Yaskawa INFORM job: DEMO_ROOF_SIDE_0625_3PAINT_45.JBI

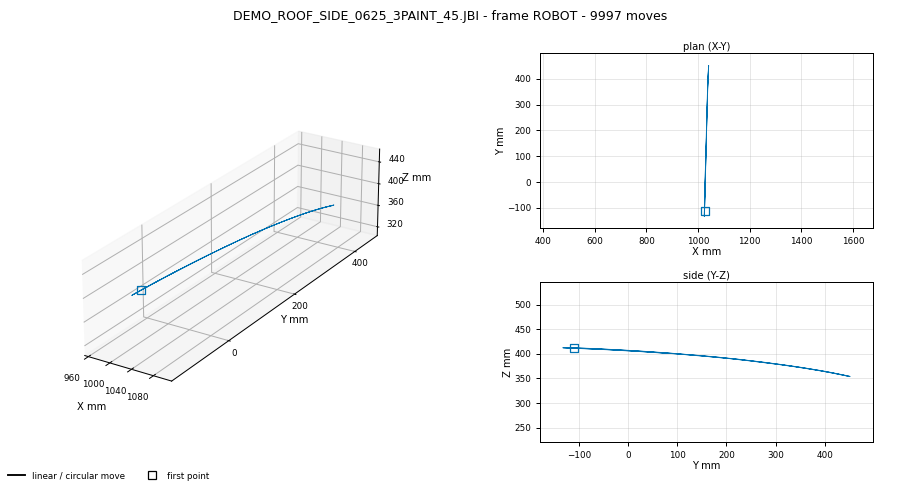
[picture p0: tool path of DEMO_ROOF_SIDE_0625_3PAINT_45.JBI in frame ROBOT, 9997 of 9997 moves have a stored position in this frame; points joined in program order, loops and branches not executed]
/JOB
//NAME DEMO_ROOF_SIDE_0625_3PAINT45
//POS
///NPOS 9997,0,0,0,0,0
///TOOL 0
///USER 0
///POSTYPE ROBOT
///RECTAN
///RCONF 1,0,0,0,0,0,0,0,0,0,0,0,0,0,0,0,0,0,0,0,0,0,0,0
C00000=1025.826,-110.558,412.586,166.562,45.746,158.343
C00001=1025.832,-110.309,412.577,166.564,45.743,158.343
C00002=1025.837,-110.058,412.568,166.568,45.740,158.343
C00003=1025.843,-109.809,412.559,166.570,45.738,158.343
C00004=1025.849,-109.559,412.550,166.574,45.735,158.343
C00005=1025.854,-109.310,412.541,166.577,45.732,158.343
C00006=1025.860,-109.059,412.532,166.579,45.729,158.343
C00007=1025.866,-108.810,412.523,166.583,45.726,158.342
C00008=1025.872,-108.560,412.514,166.586,45.724,158.342
C00009=1025.877,-108.311,412.505,166.589,45.721,158.342
C00010=1025.883,-108.060,412.496,166.592,45.718,158.342
C00011=1025.889,-107.811,412.487,166.594,45.716,158.342
C00012=1025.895,-107.561,412.478,166.598,45.713,158.342
C00013=1025.900,-107.312,412.469,166.601,45.710,158.342
C00014=1025.906,-107.061,412.460,166.604,45.708,158.341
C00015=1025.912,-106.812,412.450,166.607,45.705,158.341
C00016=1025.918,-106.562,412.442,166.609,45.703,158.341
C00017=1025.924,-106.312,412.432,166.613,45.700,158.341
C00018=1025.929,-106.063,412.423,166.616,45.697,158.341
C00019=1025.935,-105.812,412.414,166.618,45.694,158.341
C00020=1025.941,-105.563,412.405,166.622,45.692,158.341
C00021=1025.946,-105.313,412.395,166.624,45.689,158.340
C00022=1025.952,-105.063,412.386,166.628,45.686,158.340
C00023=1025.958,-104.814,412.377,166.630,45.684,158.340
C00024=1025.964,-104.564,412.367,166.634,45.681,158.340
C00025=1025.969,-104.314,412.359,166.637,45.678,158.340
C00026=1025.975,-104.064,412.349,166.640,45.676,158.340
C00027=1025.981,-103.814,412.339,166.643,45.673,158.340
C00028=1025.986,-103.565,412.330,166.645,45.670,158.340
C00029=1025.992,-103.315,412.321,166.649,45.668,158.340
C00030=1025.998,-103.066,412.312,166.651,45.665,158.339
C00031=1026.004,-102.816,412.302,166.654,45.662,158.339
C00032=1026.010,-102.566,412.293,166.658,45.659,158.339
C00033=1026.014,-102.316,412.283,166.660,45.657,158.339
C00034=1026.021,-102.066,412.274,166.664,45.654,158.339
C00035=1026.027,-101.817,412.264,166.666,45.652,158.339
C00036=1026.032,-101.567,412.255,166.670,45.649,158.339
C00037=1026.039,-101.281,412.244,166.673,45.646,158.338
C00038=1026.046,-100.994,412.233,166.676,45.643,158.338
C00039=1026.052,-100.708,412.223,166.679,45.640,158.338
C00040=1026.059,-100.422,412.211,166.683,45.637,158.338
C00041=1026.064,-100.173,412.203,166.686,45.634,158.338
C00042=1026.070,-99.923,412.193,166.690,45.631,158.338
C00043=1026.077,-99.673,412.184,166.692,45.629,158.337
C00044=1026.083,-99.423,412.174,166.696,45.626,158.337
C00045=1026.088,-99.174,412.164,166.698,45.624,158.337
C00046=1026.094,-98.924,412.155,166.701,45.621,158.337
C00047=1026.100,-98.674,412.145,166.704,45.619,158.337
C00048=1026.106,-98.424,412.136,166.707,45.616,158.337
C00049=1026.111,-98.175,412.127,166.711,45.613,158.337
C00050=1026.117,-97.925,412.117,166.713,45.610,158.336
C00051=1026.123,-97.675,412.107,166.716,45.608,158.336
C00052=1026.129,-97.425,412.098,166.719,45.605,158.336
C00053=1026.134,-97.176,412.088,166.722,45.603,158.336
C00054=1026.140,-96.926,412.078,166.725,45.600,158.336
C00055=1026.146,-96.676,412.068,166.728,45.598,158.336
C00056=1026.152,-96.426,412.059,166.731,45.595,158.336
C00057=1026.157,-96.176,412.049,166.734,45.593,158.336
C00058=1026.163,-95.927,412.039,166.737,45.590,158.336
C00059=1026.168,-95.677,412.028,166.740,45.588,158.336
C00060=1026.175,-95.427,412.019,166.742,45.585,158.335
C00061=1026.179,-95.178,412.009,166.746,45.583,158.335
C00062=1026.186,-94.928,411.999,166.748,45.580,158.335
C00063=1026.192,-94.678,411.990,166.752,45.577,158.335
C00064=1026.197,-94.428,411.980,166.754,45.575,158.335
C00065=1026.203,-94.178,411.970,166.758,45.572,158.335
C00066=1026.208,-93.929,411.960,166.760,45.570,158.335
C00067=1026.214,-93.679,411.951,166.764,45.567,158.334
C00068=1026.220,-93.430,411.940,166.766,45.565,158.334
C00069=1026.226,-93.180,411.930,166.770,45.562,158.334
C00070=1026.232,-92.930,411.920,166.772,45.560,158.334
C00071=1026.238,-92.680,411.911,166.775,45.557,158.334
C00072=1026.243,-92.431,411.901,166.778,45.555,158.334
C00073=1026.249,-92.182,411.891,166.781,45.552,158.334
C00074=1026.255,-91.931,411.880,166.785,45.550,158.334
C00075=1026.261,-91.682,411.871,166.787,45.547,158.334
C00076=1026.266,-91.431,411.861,166.791,45.545,158.334
C00077=1026.272,-91.182,411.851,166.793,45.542,158.333
C00078=1026.278,-90.932,411.840,166.797,45.539,158.333
C00079=1026.284,-90.682,411.831,166.799,45.537,158.333
C00080=1026.289,-90.433,411.821,166.802,45.534,158.333
C00081=1026.295,-90.183,411.811,166.805,45.532,158.333
C00082=1026.301,-89.934,411.800,166.808,45.529,158.333
C00083=1026.307,-89.684,411.791,166.811,45.527,158.333
C00084=1026.313,-89.434,411.781,166.814,45.524,158.332
C00085=1026.319,-89.185,411.770,166.817,45.522,158.332
C00086=1026.325,-88.935,411.760,166.820,45.519,158.332
C00087=1026.331,-88.685,411.751,166.823,45.516,158.332
C00088=1026.336,-88.435,411.740,166.826,45.514,158.332
C00089=1026.343,-88.185,411.730,166.828,45.512,158.332
C00090=1026.348,-87.935,411.720,166.832,45.509,158.332
C00091=1026.354,-87.686,411.710,166.834,45.507,158.332
C00092=1026.360,-87.436,411.700,166.838,45.504,158.332
C00093=1026.366,-87.186,411.690,166.840,45.502,158.331
C00094=1026.372,-86.937,411.679,166.844,45.499,158.331
C00095=1026.377,-86.687,411.669,166.846,45.497,158.331
C00096=1026.384,-86.437,411.659,166.850,45.494,158.331
C00097=1026.389,-86.187,411.649,166.852,45.492,158.331
C00098=1026.395,-85.938,411.639,166.856,45.489,158.331
C00099=1026.401,-85.688,411.628,166.858,45.487,158.331
C00100=1026.407,-85.438,411.619,166.861,45.484,158.330
C00101=1026.414,-85.154,411.607,166.865,45.481,158.330
C00102=1026.420,-84.871,411.596,166.868,45.478,158.330
C00103=1026.427,-84.586,411.584,166.871,45.475,158.330
C00104=1026.434,-84.303,411.572,166.875,45.472,158.330
C00105=1026.440,-84.053,411.562,166.877,45.470,158.330
C00106=1026.445,-83.803,411.551,166.881,45.467,158.330
C00107=1026.452,-83.554,411.542,166.884,45.465,158.330
C00108=1026.458,-83.303,411.531,166.887,45.462,158.329
C00109=1026.464,-83.054,411.521,166.890,45.459,158.329
C00110=1026.470,-82.804,411.510,166.893,45.457,158.329
C00111=1026.476,-82.554,411.501,166.896,45.454,158.329
C00112=1026.482,-82.305,411.490,166.899,45.452,158.329
C00113=1026.488,-82.055,411.480,166.902,45.449,158.329
C00114=1026.494,-81.806,411.469,166.904,45.446,158.328
C00115=1026.499,-81.556,411.459,166.908,45.444,158.328
C00116=1026.506,-81.306,411.449,166.910,45.441,158.328
C00117=1026.511,-81.056,411.439,166.914,45.439,158.328
C00118=1026.518,-80.806,411.428,166.916,45.436,158.328
C00119=1026.524,-80.557,411.417,166.919,45.433,158.328
C00120=1026.530,-80.307,411.408,166.922,45.431,158.328
C00121=1026.536,-80.058,411.397,166.925,45.428,158.328
C00122=1026.541,-79.807,411.386,166.928,45.426,158.327
C00123=1026.547,-79.558,411.376,166.931,45.424,158.327
C00124=1026.553,-79.309,411.365,166.934,45.421,158.327
C00125=1026.559,-79.058,411.355,166.937,45.419,158.327
C00126=1026.565,-78.808,411.344,166.940,45.417,158.327
C00127=1026.571,-78.559,411.333,166.943,45.414,158.327
C00128=1026.577,-78.310,411.322,166.946,45.412,158.327
C00129=1026.582,-78.059,411.312,166.948,45.410,158.327
C00130=1026.589,-77.810,411.302,166.952,45.407,158.326
C00131=1026.595,-77.560,411.290,166.954,45.405,158.326
C00132=1026.601,-77.311,411.280,166.958,45.402,158.326
C00133=1026.606,-77.061,411.269,166.960,45.400,158.326
C00134=1026.612,-76.811,411.259,166.963,45.397,158.326
C00135=1026.618,-76.561,411.248,166.966,45.395,158.326
C00136=1026.624,-76.312,411.237,166.970,45.392,158.326
C00137=1026.630,-76.062,411.226,166.972,45.390,158.326
C00138=1026.636,-75.813,411.215,166.976,45.387,158.326
C00139=1026.642,-75.562,411.205,166.978,45.385,158.325
C00140=1026.647,-75.313,411.194,166.980,45.383,158.325
C00141=1026.653,-75.064,411.183,166.984,45.380,158.325
C00142=1026.660,-74.814,411.173,166.986,45.378,158.325
C00143=1026.666,-74.564,411.162,166.990,45.375,158.325
C00144=1026.672,-74.315,411.151,166.992,45.373,158.325
C00145=1026.677,-74.065,411.140,166.996,45.371,158.325
C00146=1026.684,-73.815,411.129,166.998,45.368,158.325
C00147=1026.689,-73.565,411.119,167.001,45.366,158.324
C00148=1026.694,-73.315,411.107,167.004,45.364,158.324
C00149=1026.700,-73.066,411.096,167.007,45.362,158.324
C00150=1026.706,-72.815,411.085,167.009,45.359,158.324
C00151=1026.712,-72.566,411.074,167.013,45.357,158.324
C00152=1026.718,-72.316,411.063,167.016,45.355,158.324
C00153=1026.724,-72.068,411.052,167.019,45.352,158.324
C00154=1026.730,-71.817,411.040,167.021,45.350,158.324
C00155=1026.736,-71.568,411.030,167.024,45.348,158.324
C00156=1026.741,-71.318,411.018,167.028,45.345,158.324
C00157=1026.747,-71.068,411.007,167.030,45.343,158.323
C00158=1026.753,-70.818,410.996,167.033,45.341,158.323
C00159=1026.759,-70.569,410.985,167.036,45.338,158.323
C00160=1026.764,-70.319,410.974,167.039,45.336,158.323
C00161=1026.771,-70.069,410.963,167.042,45.333,158.323
C00162=1026.776,-69.820,410.952,167.045,45.331,158.323
C00163=1026.782,-69.570,410.941,167.047,45.329,158.323
C00164=1026.788,-69.320,410.929,167.051,45.326,158.323
C00165=1026.795,-69.039,410.917,167.054,45.324,158.323
C00166=1026.801,-68.757,410.904,167.056,45.322,158.323
C00167=1026.808,-68.475,410.892,167.060,45.319,158.322
C00168=1026.814,-68.193,410.879,167.063,45.316,158.322
C00169=1026.821,-67.944,410.867,167.066,45.314,158.322
C00170=1026.827,-67.694,410.857,167.069,45.311,158.322
C00171=1026.832,-67.445,410.846,167.072,45.309,158.322
C00172=1026.838,-67.194,410.834,167.075,45.307,158.322
C00173=1026.844,-66.945,410.823,167.078,45.305,158.322
C00174=1026.850,-66.695,410.811,167.080,45.302,158.322
C00175=1026.856,-66.445,410.800,167.084,45.300,158.322
C00176=1026.862,-66.196,410.789,167.087,45.298,158.322
C00177=1026.868,-65.946,410.778,167.089,45.296,158.321
C00178=1026.874,-65.697,410.766,167.093,45.293,158.321
C00179=1026.880,-65.446,410.755,167.095,45.291,158.321
C00180=1026.885,-65.197,410.744,167.097,45.289,158.321
C00181=1026.891,-64.947,410.733,167.101,45.286,158.321
C00182=1026.898,-64.698,410.721,167.104,45.284,158.321
C00183=1026.904,-64.448,410.710,167.107,45.281,158.321
C00184=1026.910,-64.198,410.699,167.110,45.279,158.321
C00185=1026.915,-63.949,410.687,167.112,45.277,158.320
C00186=1026.922,-63.699,410.675,167.116,45.274,158.320
C00187=1026.927,-63.449,410.664,167.118,45.272,158.320
C00188=1026.933,-63.200,410.653,167.121,45.270,158.320
C00189=1026.940,-62.950,410.642,167.124,45.268,158.320
C00190=1026.945,-62.700,410.630,167.127,45.266,158.320
C00191=1026.951,-62.451,410.618,167.130,45.263,158.320
C00192=1026.957,-62.201,410.607,167.133,45.261,158.320
C00193=1026.963,-61.951,410.596,167.135,45.259,158.320
C00194=1026.969,-61.702,410.584,167.138,45.256,158.319
C00195=1026.976,-61.452,410.573,167.141,45.254,158.319
C00196=1026.981,-61.202,410.562,167.144,45.252,158.319
C00197=1026.987,-60.953,410.550,167.147,45.249,158.319
C00198=1026.993,-60.703,410.539,167.150,45.247,158.319
C00199=1027.000,-60.454,410.527,167.152,45.245,158.319
C00200=1027.006,-60.204,410.516,167.156,45.242,158.319
C00201=1027.011,-59.954,410.503,167.158,45.240,158.319
C00202=1027.018,-59.704,410.492,167.162,45.238,158.319
C00203=1027.024,-59.455,410.481,167.164,45.235,158.318
C00204=1027.030,-59.205,410.469,167.167,45.233,158.318
C00205=1027.036,-58.956,410.459,167.170,45.230,158.318
C00206=1027.042,-58.706,410.446,167.173,45.228,158.318
C00207=1027.048,-58.456,410.435,167.175,45.226,158.318
C00208=1027.054,-58.207,410.423,167.178,45.223,158.318
C00209=1027.061,-57.956,410.412,167.181,45.221,158.318
C00210=1027.066,-57.707,410.400,167.185,45.219,158.318
C00211=1027.072,-57.457,410.388,167.187,45.216,158.317
C00212=1027.078,-57.208,410.377,167.190,45.214,158.317
C00213=1027.085,-56.958,410.366,167.193,45.211,158.317
C00214=1027.091,-56.708,410.354,167.195,45.209,158.317
C00215=1027.097,-56.459,410.341,167.198,45.207,158.317
C00216=1027.103,-56.209,410.330,167.201,45.204,158.317
C00217=1027.109,-55.960,410.319,167.204,45.202,158.317
C00218=1027.115,-55.710,410.307,167.207,45.199,158.316
C00219=1027.122,-55.460,410.295,167.210,45.197,158.316
C00220=1027.127,-55.211,410.284,167.213,45.195,158.316
C00221=1027.134,-54.961,410.272,167.216,45.192,158.316
C00222=1027.140,-54.712,410.260,167.218,45.190,158.316
C00223=1027.146,-54.462,410.249,167.221,45.188,158.316
C00224=1027.152,-54.212,410.237,167.224,45.185,158.316
C00225=1027.158,-53.962,410.225,167.227,45.183,158.316
C00226=1027.164,-53.713,410.214,167.229,45.181,158.315
C00227=1027.171,-53.464,410.202,167.233,45.179,158.315
C00228=1027.177,-53.213,410.190,167.235,45.176,158.315
C00229=1027.183,-52.933,410.177,167.239,45.174,158.315
C00230=1027.191,-52.652,410.164,167.242,45.171,158.315
C00231=1027.197,-52.372,410.150,167.246,45.168,158.315
C00232=1027.205,-52.091,410.137,167.248,45.165,158.315
C00233=1027.211,-51.842,410.126,167.252,45.163,158.314
C00234=1027.217,-51.592,410.114,167.254,45.160,158.314
C00235=1027.223,-51.342,410.101,167.256,45.158,158.314
C00236=1027.230,-51.092,410.090,167.260,45.156,158.314
C00237=1027.236,-50.843,410.078,167.262,45.153,158.314
C00238=1027.241,-50.593,410.066,167.266,45.151,158.314
C00239=1027.248,-50.344,410.054,167.269,45.149,158.314
C00240=1027.254,-50.093,410.042,167.271,45.146,158.314
C00241=1027.259,-49.844,410.030,167.273,45.144,158.313
C00242=1027.266,-49.594,410.018,167.277,45.142,158.313
C00243=1027.272,-49.345,410.005,167.280,45.140,158.313
C00244=1027.278,-49.095,409.993,167.282,45.138,158.313
C00245=1027.284,-48.846,409.981,167.285,45.136,158.313
C00246=1027.289,-48.596,409.969,167.288,45.133,158.313
C00247=1027.296,-48.346,409.957,167.291,45.131,158.313
C00248=1027.302,-48.096,409.944,167.293,45.129,158.313
C00249=1027.308,-47.848,409.933,167.296,45.127,158.313
C00250=1027.314,-47.598,409.920,167.299,45.125,158.313
C00251=1027.320,-47.348,409.907,167.302,45.122,158.312
C00252=1027.326,-47.098,409.895,167.304,45.120,158.312
C00253=1027.332,-46.849,409.883,167.307,45.118,158.312
C00254=1027.338,-46.599,409.871,167.311,45.116,158.312
C00255=1027.344,-46.350,409.859,167.313,45.113,158.312
C00256=1027.350,-46.100,409.846,167.316,45.111,158.312
C00257=1027.356,-45.850,409.834,167.319,45.109,158.312
C00258=1027.362,-45.601,409.822,167.322,45.107,158.312
C00259=1027.368,-45.351,409.809,167.324,45.105,158.312
C00260=1027.375,-45.102,409.798,167.327,45.103,158.311
C00261=1027.381,-44.852,409.785,167.330,45.100,158.311
C00262=1027.387,-44.602,409.772,167.333,45.098,158.311
C00263=1027.393,-44.352,409.760,167.335,45.096,158.311
C00264=1027.399,-44.103,409.748,167.338,45.094,158.311
C00265=1027.404,-43.853,409.736,167.341,45.091,158.311
C00266=1027.411,-43.604,409.724,167.344,45.089,158.311
C00267=1027.417,-43.354,409.711,167.346,45.087,158.311
C00268=1027.423,-43.104,409.699,167.349,45.085,158.310
C00269=1027.430,-42.854,409.687,167.352,45.083,158.310
C00270=1027.436,-42.605,409.673,167.355,45.081,158.310
C00271=1027.441,-42.356,409.661,167.358,45.079,158.310
C00272=1027.448,-42.106,409.649,167.360,45.076,158.310
C00273=1027.454,-41.856,409.637,167.364,45.074,158.310
C00274=1027.460,-41.606,409.624,167.366,45.072,158.310
C00275=1027.466,-41.357,409.612,167.369,45.070,158.310
C00276=1027.472,-41.107,409.600,167.371,45.067,158.309
C00277=1027.478,-40.858,409.586,167.375,45.065,158.309
C00278=1027.485,-40.608,409.574,167.377,45.063,158.309
C00279=1027.491,-40.358,409.562,167.380,45.061,158.309
C00280=1027.497,-40.108,409.549,167.382,45.058,158.309
C00281=1027.503,-39.859,409.537,167.386,45.056,158.309
C00282=1027.509,-39.610,409.524,167.388,45.054,158.309
C00283=1027.515,-39.360,409.512,167.391,45.051,158.309
C00284=1027.522,-39.111,409.500,167.394,45.049,158.309
C00285=1027.528,-38.861,409.487,167.397,45.047,158.308
C00286=1027.534,-38.612,409.474,167.399,45.045,158.308
C00287=1027.540,-38.362,409.462,167.402,45.043,158.308
C00288=1027.546,-38.112,409.449,167.405,45.041,158.308
C00289=1027.551,-37.862,409.436,167.408,45.038,158.308
C00290=1027.558,-37.613,409.423,167.411,45.036,158.308
C00291=1027.564,-37.363,409.411,167.413,45.034,158.308
C00292=1027.570,-37.114,409.397,167.416,45.032,158.308
C00293=1027.577,-36.833,409.383,167.419,45.030,158.308
C00294=1027.584,-36.553,409.369,167.422,45.027,158.307
C00295=1027.590,-36.273,409.355,167.425,45.025,158.307
C00296=1027.597,-35.993,409.340,167.428,45.023,158.307
C00297=1027.603,-35.743,409.327,167.431,45.020,158.307
C00298=1027.610,-35.494,409.315,167.434,45.018,158.307
C00299=1027.616,-35.244,409.302,167.436,45.016,158.307
C00300=1027.622,-34.994,409.290,167.439,45.014,158.307
C00301=1027.628,-34.745,409.276,167.442,45.012,158.307
C00302=1027.634,-34.495,409.264,167.445,45.010,158.307
C00303=1027.640,-34.246,409.251,167.447,45.007,158.306
C00304=1027.646,-33.996,409.238,167.450,45.005,158.306
C00305=1027.652,-33.747,409.225,167.453,45.003,158.306
C00306=1027.658,-33.497,409.212,167.455,45.001,158.306
C00307=1027.664,-33.247,409.199,167.458,44.999,158.306
C00308=1027.670,-32.998,409.186,167.461,44.997,158.306
C00309=1027.676,-32.748,409.173,167.464,44.995,158.306
C00310=1027.682,-32.498,409.161,167.466,44.993,158.306
C00311=1027.688,-32.249,409.147,167.469,44.991,158.306
C00312=1027.695,-31.999,409.134,167.471,44.989,158.305
C00313=1027.701,-31.749,409.121,167.475,44.986,158.305
C00314=1027.707,-31.499,409.109,167.477,44.984,158.305
C00315=1027.713,-31.250,409.095,167.480,44.982,158.305
C00316=1027.719,-31.001,409.082,167.483,44.980,158.305
C00317=1027.726,-30.751,409.070,167.485,44.978,158.305
C00318=1027.732,-30.502,409.057,167.489,44.976,158.305
C00319=1027.738,-30.252,409.044,167.491,44.973,158.305
C00320=1027.744,-30.003,409.031,167.494,44.971,158.304
C00321=1027.750,-29.753,409.018,167.496,44.969,158.304
C00322=1027.757,-29.503,409.005,167.499,44.967,158.304
C00323=1027.763,-29.254,408.992,167.501,44.965,158.304
C00324=1027.769,-29.004,408.979,167.505,44.962,158.304
C00325=1027.775,-28.755,408.966,167.507,44.960,158.304
C00326=1027.782,-28.505,408.952,167.510,44.958,158.304
C00327=1027.788,-28.255,408.940,167.513,44.956,158.304
C00328=1027.794,-28.006,408.927,167.515,44.953,158.303
C00329=1027.801,-27.756,408.913,167.518,44.951,158.303
C00330=1027.806,-27.506,408.900,167.521,44.949,158.303
C00331=1027.813,-27.257,408.887,167.524,44.947,158.303
C00332=1027.819,-27.008,408.874,167.526,44.945,158.303
C00333=1027.824,-26.758,408.861,167.529,44.943,158.303
C00334=1027.830,-26.508,408.847,167.531,44.941,158.303
C00335=1027.837,-26.258,408.834,167.534,44.939,158.303
C00336=1027.843,-26.009,408.821,167.536,44.937,158.303
C00337=1027.849,-25.760,408.807,167.540,44.934,158.302
C00338=1027.855,-25.510,408.794,167.543,44.932,158.302
C00339=1027.861,-25.260,408.781,167.545,44.930,158.302
C00340=1027.867,-25.011,408.768,167.548,44.928,158.302
C00341=1027.873,-24.761,408.753,167.550,44.926,158.302
C00342=1027.879,-24.512,408.740,167.553,44.925,158.302
C00343=1027.886,-24.262,408.727,167.555,44.923,158.302
C00344=1027.892,-24.012,408.714,167.558,44.921,158.302
C00345=1027.897,-23.763,408.700,167.561,44.919,158.302
C00346=1027.904,-23.513,408.687,167.564,44.916,158.302
C00347=1027.910,-23.264,408.674,167.567,44.914,158.301
C00348=1027.916,-23.014,408.660,167.569,44.912,158.301
C00349=1027.922,-22.765,408.646,167.572,44.910,158.301
C00350=1027.928,-22.516,408.633,167.574,44.908,158.301
C00351=1027.935,-22.266,408.619,167.577,44.906,158.301
C00352=1027.941,-22.016,408.606,167.579,44.904,158.301
C00353=1027.946,-21.767,408.592,167.582,44.902,158.301
C00354=1027.953,-21.518,408.579,167.585,44.900,158.301
C00355=1027.959,-21.267,408.566,167.588,44.898,158.301
C00356=1027.965,-21.018,408.553,167.591,44.895,158.300
C00357=1027.972,-20.737,408.537,167.593,44.893,158.300
C00358=1027.979,-20.455,408.521,167.597,44.891,158.300
C00359=1027.986,-20.175,408.507,167.599,44.888,158.300
C00360=1027.993,-19.894,408.492,167.603,44.886,158.300
C00361=1027.999,-19.644,408.478,167.605,44.884,158.300
C00362=1028.006,-19.394,408.465,167.608,44.881,158.300
C00363=1028.011,-19.145,408.451,167.610,44.879,158.299
C00364=1028.018,-18.896,408.438,167.613,44.877,158.299
C00365=1028.024,-18.646,408.424,167.615,44.875,158.299
C00366=1028.030,-18.396,408.410,167.618,44.873,158.299
C00367=1028.036,-18.147,408.397,167.622,44.871,158.299
C00368=1028.043,-17.897,408.383,167.624,44.869,158.299
C00369=1028.049,-17.648,408.370,167.627,44.867,158.299
C00370=1028.055,-17.398,408.356,167.629,44.865,158.299
C00371=1028.061,-17.148,408.342,167.632,44.863,158.298
C00372=1028.068,-16.899,408.328,167.634,44.861,158.298
C00373=1028.073,-16.650,408.315,167.637,44.859,158.298
C00374=1028.080,-16.400,408.301,167.639,44.856,158.298
C00375=1028.087,-16.151,408.288,167.642,44.854,158.298
C00376=1028.093,-15.901,408.274,167.645,44.852,158.298
C00377=1028.099,-15.651,408.260,167.648,44.850,158.298
C00378=1028.105,-15.402,408.247,167.651,44.848,158.298
C00379=1028.111,-15.151,408.233,167.653,44.846,158.298
C00380=1028.118,-14.903,408.219,167.656,44.844,158.297
C00381=1028.123,-14.653,408.205,167.658,44.842,158.297
C00382=1028.130,-14.403,408.191,167.661,44.840,158.297
C00383=1028.135,-14.154,408.177,167.663,44.838,158.297
C00384=1028.142,-13.904,408.164,167.666,44.836,158.297
C00385=1028.148,-13.655,408.149,167.669,44.834,158.297
C00386=1028.153,-13.405,408.135,167.671,44.832,158.297
C00387=1028.160,-13.155,408.122,167.674,44.829,158.297
C00388=1028.166,-12.906,408.107,167.676,44.827,158.296
C00389=1028.172,-12.657,408.094,167.679,44.825,158.296
C00390=1028.178,-12.407,408.079,167.681,44.824,158.296
C00391=1028.185,-12.157,408.066,167.684,44.822,158.296
C00392=1028.191,-11.908,408.051,167.687,44.820,158.296
C00393=1028.197,-11.659,408.038,167.689,44.818,158.296
C00394=1028.203,-11.408,408.024,167.692,44.816,158.296
C00395=1028.210,-11.160,408.010,167.694,44.814,158.296
C00396=1028.215,-10.910,407.996,167.697,44.812,158.296
C00397=1028.221,-10.660,407.982,167.699,44.810,158.295
C00398=1028.228,-10.411,407.968,167.703,44.808,158.295
C00399=1028.234,-10.161,407.953,167.706,44.806,158.295
C00400=1028.240,-9.912,407.939,167.708,44.804,158.295
C00401=1028.247,-9.662,407.925,167.711,44.801,158.295
C00402=1028.253,-9.413,407.912,167.713,44.799,158.295
C00403=1028.259,-9.163,407.897,167.716,44.797,158.295
C00404=1028.265,-8.913,407.883,167.718,44.795,158.295
C00405=1028.271,-8.663,407.870,167.721,44.793,158.295
C00406=1028.277,-8.415,407.855,167.723,44.791,158.294
C00407=1028.284,-8.165,407.841,167.726,44.789,158.294
C00408=1028.290,-7.916,407.827,167.729,44.787,158.294
C00409=1028.297,-7.666,407.813,167.731,44.785,158.294
C00410=1028.302,-7.417,407.799,167.734,44.783,158.294
C00411=1028.308,-7.166,407.784,167.736,44.781,158.294
C00412=1028.315,-6.918,407.770,167.739,44.779,158.294
C00413=1028.321,-6.667,407.756,167.741,44.777,158.294
C00414=1028.327,-6.418,407.743,167.744,44.775,158.293
C00415=1028.334,-6.169,407.728,167.747,44.773,158.293
C00416=1028.340,-5.919,407.715,167.749,44.771,158.293
C00417=1028.346,-5.670,407.700,167.751,44.768,158.293
C00418=1028.352,-5.420,407.686,167.754,44.766,158.293
C00419=1028.359,-5.171,407.671,167.757,44.764,158.293
C00420=1028.364,-4.921,407.658,167.759,44.762,158.293
C00421=1028.372,-4.639,407.641,167.763,44.760,158.293
C00422=1028.379,-4.356,407.625,167.765,44.757,158.292
C00423=1028.386,-4.072,407.609,167.769,44.755,158.292
C00424=1028.394,-3.791,407.593,167.771,44.752,158.292
C00425=1028.399,-3.542,407.578,167.774,44.751,158.292
C00426=1028.405,-3.291,407.564,167.776,44.749,158.292
C00427=1028.412,-3.042,407.549,167.779,44.747,158.292
C00428=1028.418,-2.793,407.534,167.782,44.745,158.292
C00429=1028.424,-2.542,407.520,167.784,44.743,158.292
C00430=1028.429,-2.293,407.506,167.787,44.741,158.291
C00431=1028.436,-2.044,407.491,167.789,44.739,158.291
C00432=1028.441,-1.794,407.477,167.792,44.737,158.291
C00433=1028.448,-1.545,407.462,167.795,44.735,158.291
C00434=1028.454,-1.296,407.448,167.797,44.734,158.291
C00435=1028.461,-1.046,407.433,167.800,44.732,158.291
C00436=1028.467,-0.796,407.419,167.802,44.730,158.291
C00437=1028.472,-0.547,407.404,167.805,44.728,158.291
C00438=1028.479,-0.297,407.389,167.808,44.726,158.291
C00439=1028.485,-0.048,407.374,167.810,44.724,158.290
C00440=1028.491,0.202,407.360,167.812,44.722,158.290
C00441=1028.497,0.452,407.345,167.814,44.720,158.290
C00442=1028.503,0.700,407.331,167.817,44.718,158.290
C00443=1028.509,0.950,407.316,167.819,44.716,158.290
C00444=1028.516,1.200,407.301,167.822,44.714,158.290
C00445=1028.521,1.449,407.287,167.825,44.712,158.290
C00446=1028.527,1.699,407.272,167.827,44.710,158.290
C00447=1028.533,1.948,407.257,167.830,44.708,158.290
C00448=1028.540,2.198,407.243,167.832,44.706,158.289
C00449=1028.546,2.447,407.228,167.835,44.704,158.289
C00450=1028.553,2.696,407.214,167.838,44.702,158.289
C00451=1028.559,2.946,407.199,167.840,44.700,158.289
C00452=1028.565,3.196,407.184,167.843,44.698,158.289
C00453=1028.571,3.445,407.170,167.845,44.696,158.289
C00454=1028.577,3.694,407.155,167.848,44.694,158.289
C00455=1028.584,3.944,407.140,167.851,44.692,158.289
C00456=1028.589,4.193,407.125,167.853,44.691,158.289
C00457=1028.596,4.443,407.110,167.855,44.688,158.288
C00458=1028.602,4.692,407.095,167.858,44.686,158.288
C00459=1028.608,4.942,407.081,167.861,44.684,158.288
C00460=1028.614,5.192,407.067,167.863,44.682,158.288
C00461=1028.620,5.441,407.052,167.866,44.680,158.288
C00462=1028.627,5.691,407.037,167.868,44.678,158.288
C00463=1028.632,5.940,407.022,167.870,44.676,158.288
C00464=1028.639,6.190,407.007,167.873,44.674,158.287
C00465=1028.645,6.439,406.992,167.875,44.672,158.287
C00466=1028.652,6.689,406.977,167.878,44.670,158.287
C00467=1028.657,6.938,406.963,167.880,44.668,158.287
C00468=1028.664,7.187,406.948,167.883,44.667,158.287
C00469=1028.670,7.427,406.933,167.885,44.665,158.287
C00470=1028.676,7.667,406.920,167.888,44.663,158.287
C00471=1028.682,7.907,406.905,167.891,44.661,158.287
C00472=1028.688,8.147,406.891,167.893,44.659,158.286
C00473=1028.694,8.387,406.876,167.896,44.657,158.286
C00474=1028.700,8.626,406.862,167.897,44.655,158.286
C00475=1028.706,8.866,406.848,167.900,44.653,158.286
C00476=1028.713,9.106,406.833,167.903,44.651,158.286
C00477=1028.718,9.355,406.819,167.905,44.648,158.286
C00478=1028.725,9.605,406.804,167.908,44.646,158.286
C00479=1028.731,9.855,406.789,167.910,44.644,158.285
C00480=1028.738,10.104,406.774,167.913,44.643,158.285
C00481=1028.744,10.354,406.759,167.915,44.641,158.285
C00482=1028.750,10.603,406.744,167.918,44.639,158.285
C00483=1028.756,10.853,406.729,167.920,44.637,158.285
C00484=1028.762,11.102,406.714,167.923,44.635,158.285
C00485=1028.771,11.406,406.696,167.925,44.632,158.285
C00486=1028.778,11.709,406.678,167.929,44.629,158.284
C00487=1028.786,12.014,406.660,167.932,44.627,158.284
C00488=1028.793,12.317,406.642,167.935,44.624,158.284
C00489=1028.800,12.567,406.627,167.937,44.622,158.284
C00490=1028.806,12.817,406.612,167.940,44.621,158.284
C00491=1028.813,13.066,406.596,167.942,44.619,158.284
C00492=1028.819,13.315,406.581,167.945,44.616,158.284
C00493=1028.826,13.565,406.566,167.947,44.614,158.283
C00494=1028.832,13.815,406.551,167.950,44.612,158.283
C00495=1028.837,14.064,406.536,167.953,44.610,158.283
C00496=1028.844,14.313,406.520,167.955,44.608,158.283
C00497=1028.850,14.563,406.506,167.958,44.606,158.283
C00498=1028.856,14.812,406.491,167.960,44.604,158.283
C00499=1028.862,15.062,406.475,167.962,44.602,158.283
C00500=1028.869,15.311,406.459,167.965,44.601,158.283
C00501=1028.875,15.561,406.444,167.967,44.599,158.282
C00502=1028.881,15.811,406.429,167.970,44.597,158.282
C00503=1028.887,16.059,406.414,167.972,44.595,158.282
C00504=1028.893,16.309,406.399,167.975,44.593,158.282
C00505=1028.900,16.558,406.384,167.977,44.591,158.282
C00506=1028.906,16.808,406.367,167.980,44.589,158.282
C00507=1028.912,17.058,406.353,167.983,44.587,158.282
C00508=1028.918,17.307,406.338,167.985,44.585,158.282
C00509=1028.925,17.556,406.322,167.987,44.583,158.281
C00510=1028.931,17.806,406.306,167.989,44.581,158.281
C00511=1028.937,18.055,406.291,167.992,44.579,158.281
C00512=1028.943,18.304,406.276,167.995,44.577,158.281
C00513=1028.949,18.554,406.261,167.997,44.575,158.281
C00514=1028.956,18.803,406.245,168.000,44.573,158.281
C00515=1028.962,19.053,406.230,168.002,44.571,158.281
C00516=1028.968,19.302,406.215,168.005,44.569,158.280
C00517=1028.974,19.552,406.199,168.007,44.567,158.280
C00518=1028.981,19.801,406.184,168.009,44.565,158.280
C00519=1028.987,20.051,406.168,168.011,44.563,158.280
C00520=1028.993,20.300,406.153,168.014,44.561,158.280
C00521=1029.000,20.550,406.137,168.017,44.559,158.280
C00522=1029.005,20.799,406.121,168.019,44.557,158.280
C00523=1029.012,21.049,406.106,168.022,44.555,158.280
C00524=1029.018,21.299,406.090,168.024,44.553,158.279
C00525=1029.024,21.548,406.075,168.027,44.551,158.279
C00526=1029.030,21.798,406.059,168.029,44.550,158.279
C00527=1029.037,22.047,406.043,168.031,44.548,158.279
C00528=1029.043,22.296,406.028,168.034,44.546,158.279
C00529=1029.049,22.546,406.012,168.036,44.544,158.279
C00530=1029.056,22.795,405.996,168.039,44.542,158.279
C00531=1029.061,23.045,405.981,168.041,44.540,158.279
C00532=1029.068,23.294,405.965,168.044,44.538,158.278
C00533=1029.074,23.544,405.950,168.047,44.536,158.278
C00534=1029.080,23.793,405.934,168.048,44.534,158.278
C00535=1029.087,24.042,405.919,168.051,44.532,158.278
C00536=1029.093,24.292,405.903,168.053,44.530,158.278
C00537=1029.099,24.541,405.887,168.056,44.528,158.278
C00538=1029.105,24.791,405.872,168.059,44.527,158.278
C00539=1029.112,25.040,405.856,168.061,44.525,158.278
C00540=1029.117,25.290,405.840,168.064,44.523,158.277
C00541=1029.124,25.539,405.825,168.066,44.521,158.277
C00542=1029.131,25.788,405.809,168.068,44.518,158.277
C00543=1029.136,26.038,405.794,168.070,44.516,158.277
C00544=1029.143,26.287,405.778,168.073,44.514,158.277
C00545=1029.149,26.536,405.762,168.075,44.512,158.277
C00546=1029.155,26.786,405.747,168.078,44.510,158.277
C00547=1029.161,27.035,405.730,168.081,44.509,158.276
C00548=1029.167,27.284,405.714,168.083,44.507,158.276
C00549=1029.175,27.570,405.696,168.086,44.505,158.276
C00550=1029.182,27.856,405.679,168.088,44.502,158.276
C00551=1029.189,28.142,405.660,168.092,44.500,158.276
C00552=1029.196,28.428,405.642,168.094,44.498,158.276
C00553=1029.203,28.677,405.626,168.097,44.496,158.276
C00554=1029.208,28.927,405.611,168.099,44.494,158.275
C00555=1029.214,29.177,405.594,168.101,44.492,158.275
C00556=1029.221,29.426,405.579,168.104,44.490,158.275
C00557=1029.227,29.675,405.562,168.106,44.488,158.275
C00558=1029.233,29.924,405.546,168.109,44.486,158.275
C00559=1029.240,30.173,405.530,168.112,44.485,158.275
C00560=1029.245,30.423,405.515,168.113,44.483,158.275
C00561=1029.251,30.673,405.499,168.116,44.481,158.275
C00562=1029.259,30.922,405.483,168.118,44.479,158.274
C00563=1029.265,31.172,405.466,168.121,44.477,158.274
C00564=1029.270,31.421,405.450,168.123,44.475,158.274
C00565=1029.277,31.670,405.434,168.126,44.473,158.274
C00566=1029.283,31.920,405.418,168.128,44.471,158.274
C00567=1029.289,32.169,405.402,168.130,44.469,158.274
C00568=1029.295,32.419,405.386,168.133,44.467,158.274
C00569=1029.301,32.668,405.371,168.135,44.466,158.274
C00570=1029.308,32.918,405.354,168.138,44.464,158.273
C00571=1029.314,33.167,405.338,168.141,44.462,158.273
C00572=1029.321,33.416,405.322,168.142,44.460,158.273
C00573=1029.327,33.666,405.306,168.145,44.458,158.273
C00574=1029.332,33.915,405.290,168.147,44.456,158.273
C00575=1029.339,34.164,405.274,168.150,44.454,158.273
C00576=1029.345,34.413,405.258,168.153,44.452,158.273
C00577=1029.352,34.663,405.241,168.155,44.450,158.272
C00578=1029.358,34.913,405.225,168.158,44.448,158.272
C00579=1029.364,35.162,405.209,168.159,44.447,158.272
C00580=1029.370,35.411,405.193,168.162,44.444,158.272
C00581=1029.376,35.661,405.177,168.164,44.442,158.272
C00582=1029.384,35.910,405.161,168.167,44.440,158.272
C00583=1029.389,36.160,405.144,168.169,44.438,158.272
C00584=1029.395,36.409,405.128,168.172,44.436,158.271
C00585=1029.402,36.658,405.112,168.174,44.434,158.271
C00586=1029.408,36.907,405.096,168.176,44.432,158.271
C00587=1029.415,37.157,405.080,168.179,44.431,158.271
C00588=1029.421,37.407,405.063,168.181,44.429,158.271
C00589=1029.427,37.656,405.047,168.184,44.427,158.271
C00590=1029.432,37.905,405.031,168.187,44.425,158.271
C00591=1029.438,38.155,405.015,168.188,44.423,158.270
C00592=1029.445,38.405,404.998,168.191,44.421,158.270
C00593=1029.451,38.654,404.982,168.193,44.419,158.270
C00594=1029.458,38.903,404.965,168.196,44.417,158.270
C00595=1029.464,39.152,404.949,168.198,44.415,158.270
C00596=1029.470,39.401,404.933,168.200,44.414,158.270
C00597=1029.476,39.651,404.916,168.203,44.412,158.270
C00598=1029.482,39.901,404.900,168.205,44.410,158.270
C00599=1029.488,40.150,404.884,168.208,44.408,158.269
C00600=1029.495,40.399,404.867,168.210,44.406,158.269
C00601=1029.501,40.649,404.850,168.212,44.404,158.269
C00602=1029.507,40.898,404.834,168.215,44.402,158.269
C00603=1029.513,41.148,404.818,168.217,44.400,158.269
C00604=1029.519,41.397,404.801,168.220,44.398,158.269
C00605=1029.526,41.646,404.784,168.222,44.396,158.269
C00606=1029.532,41.896,404.768,168.224,44.395,158.268
C00607=1029.538,42.145,404.751,168.226,44.393,158.268
C00608=1029.544,42.394,404.735,168.229,44.391,158.268
C00609=1029.550,42.644,404.718,168.232,44.389,158.268
C00610=1029.556,42.893,404.702,168.234,44.387,158.268
C00611=1029.562,43.142,404.685,168.236,44.386,158.268
C00612=1029.569,43.391,404.668,168.239,44.384,158.268
C00613=1029.575,43.678,404.649,168.241,44.382,158.268
C00614=1029.583,43.964,404.630,168.244,44.379,158.267
C00615=1029.589,44.249,404.611,168.247,44.377,158.267
C00616=1029.596,44.535,404.592,168.250,44.375,158.267
C00617=1029.603,44.784,404.575,168.252,44.373,158.267
C00618=1029.609,45.035,404.558,168.254,44.372,158.267
C00619=1029.615,45.283,404.541,168.257,44.370,158.267
C00620=1029.621,45.533,404.525,168.259,44.368,158.267
C00621=1029.628,45.782,404.507,168.262,44.366,158.267
C00622=1029.633,46.032,404.491,168.264,44.365,158.266
C00623=1029.639,46.281,404.474,168.266,44.363,158.266
C00624=1029.645,46.530,404.457,168.269,44.361,158.266
C00625=1029.652,46.780,404.441,168.271,44.359,158.266
C00626=1029.658,47.029,404.424,168.273,44.357,158.266
C00627=1029.663,47.278,404.407,168.276,44.355,158.266
C00628=1029.670,47.528,404.390,168.278,44.353,158.266
C00629=1029.676,47.777,404.373,168.281,44.352,158.266
C00630=1029.682,48.026,404.356,168.283,44.350,158.266
C00631=1029.688,48.276,404.339,168.285,44.348,158.265
C00632=1029.694,48.525,404.322,168.288,44.346,158.265
C00633=1029.700,48.774,404.306,168.290,44.345,158.265
C00634=1029.707,49.024,404.289,168.292,44.343,158.265
C00635=1029.712,49.273,404.272,168.294,44.341,158.265
C00636=1029.718,49.522,404.255,168.297,44.339,158.265
C00637=1029.725,49.772,404.238,168.300,44.337,158.265
C00638=1029.731,50.021,404.221,168.302,44.335,158.264
C00639=1029.736,50.270,404.204,168.304,44.333,158.264
C00640=1029.743,50.520,404.187,168.306,44.331,158.264
C00641=1029.749,50.769,404.171,168.309,44.329,158.264
C00642=1029.756,51.019,404.153,168.312,44.328,158.264
C00643=1029.762,51.268,404.137,168.313,44.326,158.264
C00644=1029.768,51.517,404.120,168.316,44.324,158.264
C00645=1029.774,51.766,404.102,168.318,44.322,158.263
C00646=1029.780,52.016,404.086,168.321,44.320,158.263
C00647=1029.787,52.265,404.069,168.323,44.318,158.263
C00648=1029.793,52.515,404.052,168.325,44.316,158.263
C00649=1029.799,52.764,404.035,168.328,44.314,158.263
C00650=1029.806,53.013,404.018,168.330,44.313,158.263
C00651=1029.811,53.263,404.001,168.333,44.311,158.263
C00652=1029.818,53.512,403.983,168.335,44.310,158.263
C00653=1029.824,53.761,403.966,168.337,44.308,158.263
C00654=1029.831,54.011,403.950,168.340,44.306,158.262
C00655=1029.836,54.260,403.932,168.343,44.304,158.262
C00656=1029.842,54.509,403.916,168.345,44.302,158.262
C00657=1029.849,54.759,403.899,168.346,44.299,158.262
C00658=1029.855,55.007,403.882,168.349,44.298,158.262
C00659=1029.861,55.258,403.864,168.352,44.296,158.262
C00660=1029.867,55.507,403.847,168.354,44.294,158.261
C00661=1029.874,55.756,403.830,168.356,44.292,158.261
C00662=1029.880,56.005,403.813,168.358,44.290,158.261
C00663=1029.886,56.255,403.796,168.361,44.288,158.261
C00664=1029.892,56.504,403.779,168.364,44.286,158.261
C00665=1029.899,56.753,403.762,168.366,44.284,158.261
C00666=1029.905,57.003,403.745,168.368,44.283,158.261
C00667=1029.911,57.252,403.727,168.370,44.281,158.260
C00668=1029.918,57.501,403.710,168.373,44.279,158.260
C00669=1029.924,57.750,403.693,168.376,44.277,158.260
C00670=1029.930,58.000,403.676,168.378,44.275,158.260
C00671=1029.936,58.250,403.659,168.380,44.273,158.260
C00672=1029.943,58.498,403.642,168.382,44.271,158.260
C00673=1029.950,58.748,403.625,168.385,44.269,158.260
C00674=1029.955,58.997,403.608,168.387,44.267,158.259
C00675=1029.962,59.247,403.590,168.390,44.265,158.259
C00676=1029.968,59.496,403.573,168.392,44.264,158.259
C00677=1029.975,59.781,403.553,168.395,44.261,158.259
C00678=1029.983,60.067,403.534,168.398,44.259,158.259
C00679=1029.990,60.353,403.514,168.400,44.257,158.259
C00680=1029.998,60.638,403.494,168.403,44.254,158.258
C00681=1030.003,60.888,403.477,168.405,44.253,158.258
C00682=1030.010,61.137,403.460,168.408,44.251,158.258
C00683=1030.016,61.386,403.443,168.410,44.249,158.258
C00684=1030.022,61.636,403.425,168.413,44.247,158.258
C00685=1030.029,61.885,403.408,168.415,44.245,158.258
C00686=1030.035,62.134,403.391,168.417,44.243,158.258
C00687=1030.041,62.383,403.373,168.420,44.241,158.257
C00688=1030.047,62.633,403.356,168.422,44.239,158.257
C00689=1030.054,62.882,403.339,168.425,44.237,158.257
C00690=1030.061,63.132,403.322,168.427,44.235,158.257
C00691=1030.066,63.381,403.304,168.429,44.233,158.257
C00692=1030.073,63.630,403.287,168.431,44.231,158.257
C00693=1030.079,63.879,403.269,168.434,44.229,158.256
C00694=1030.086,64.129,403.252,168.437,44.227,158.256
C00695=1030.092,64.378,403.234,168.438,44.226,158.256
C00696=1030.097,64.627,403.216,168.441,44.224,158.256
C00697=1030.104,64.877,403.199,168.443,44.222,158.256
C00698=1030.110,65.126,403.182,168.446,44.220,158.256
C00699=1030.117,65.375,403.164,168.448,44.218,158.256
C00700=1030.123,65.625,403.146,168.450,44.216,158.255
C00701=1030.129,65.874,403.129,168.453,44.214,158.255
C00702=1030.135,66.124,403.111,168.455,44.212,158.255
C00703=1030.141,66.373,403.094,168.458,44.210,158.255
C00704=1030.148,66.621,403.076,168.460,44.209,158.255
C00705=1030.154,66.871,403.058,168.462,44.207,158.255
C00706=1030.159,67.120,403.040,168.465,44.205,158.255
C00707=1030.166,67.370,403.023,168.467,44.203,158.254
C00708=1030.172,67.619,403.005,168.469,44.202,158.254
C00709=1030.179,67.868,402.988,168.472,44.200,158.254
C00710=1030.185,68.118,402.970,168.474,44.198,158.254
C00711=1030.190,68.367,402.953,168.477,44.196,158.254
C00712=1030.197,68.616,402.934,168.479,44.194,158.254
C00713=1030.204,68.865,402.917,168.481,44.193,158.254
C00714=1030.209,69.114,402.899,168.484,44.191,158.254
C00715=1030.215,69.364,402.881,168.486,44.189,158.253
C00716=1030.222,69.614,402.864,168.488,44.187,158.253
C00717=1030.228,69.863,402.846,168.490,44.185,158.253
C00718=1030.234,70.112,402.827,168.493,44.183,158.253
C00719=1030.240,70.362,402.810,168.496,44.181,158.253
C00720=1030.246,70.610,402.793,168.497,44.180,158.253
C00721=1030.252,70.860,402.775,168.500,44.178,158.253
C00722=1030.259,71.109,402.756,168.502,44.176,158.252
C00723=1030.264,71.358,402.738,168.505,44.174,158.252
C00724=1030.271,71.608,402.721,168.507,44.173,158.252
C00725=1030.277,71.857,402.703,168.509,44.171,158.252
C00726=1030.283,72.106,402.685,168.512,44.169,158.252
C00727=1030.289,72.355,402.667,168.515,44.167,158.252
C00728=1030.295,72.605,402.649,168.516,44.165,158.252
C00729=1030.301,72.854,402.631,168.519,44.163,158.252
C00730=1030.308,73.103,402.613,168.521,44.161,158.251
C00731=1030.314,73.353,402.595,168.524,44.160,158.251
C00732=1030.321,73.602,402.577,168.526,44.158,158.251
C00733=1030.326,73.851,402.559,168.528,44.156,158.251
C00734=1030.332,74.101,402.541,168.531,44.154,158.251
C00735=1030.339,74.350,402.523,168.533,44.152,158.251
C00736=1030.345,74.599,402.506,168.535,44.150,158.251
C00737=1030.351,74.848,402.488,168.538,44.148,158.250
C00738=1030.358,75.097,402.469,168.540,44.147,158.250
C00739=1030.364,75.347,402.451,168.543,44.145,158.250
C00740=1030.369,75.596,402.433,168.545,44.143,158.250
C00741=1030.376,75.882,402.413,168.548,44.141,158.250
C00742=1030.384,76.167,402.392,168.551,44.139,158.250
C00743=1030.391,76.452,402.372,168.553,44.137,158.250
C00744=1030.398,76.737,402.351,168.556,44.134,158.249
C00745=1030.405,76.987,402.332,168.558,44.133,158.249
C00746=1030.411,77.236,402.314,168.561,44.131,158.249
C00747=1030.417,77.486,402.296,168.563,44.130,158.249
C00748=1030.423,77.734,402.278,168.565,44.128,158.249
C00749=1030.429,77.984,402.260,168.568,44.126,158.249
C00750=1030.435,78.233,402.242,168.570,44.124,158.249
C00751=1030.441,78.483,402.224,168.572,44.122,158.248
C00752=1030.447,78.731,402.205,168.574,44.120,158.248
C00753=1030.454,78.981,402.187,168.577,44.118,158.248
C00754=1030.459,79.231,402.168,168.580,44.117,158.248
C00755=1030.465,79.480,402.150,168.581,44.115,158.248
C00756=1030.471,79.729,402.132,168.584,44.113,158.248
C00757=1030.477,79.978,402.113,168.587,44.112,158.248
C00758=1030.484,80.228,402.095,168.589,44.110,158.248
C00759=1030.490,80.477,402.077,168.591,44.108,158.247
C00760=1030.496,80.726,402.058,168.593,44.106,158.247
C00761=1030.502,80.975,402.041,168.596,44.105,158.247
C00762=1030.508,81.224,402.022,168.598,44.103,158.247
C00763=1030.515,81.473,402.003,168.600,44.101,158.247
C00764=1030.520,81.723,401.985,168.603,44.099,158.247
C00765=1030.527,81.972,401.966,168.606,44.097,158.247
C00766=1030.532,82.221,401.948,168.607,44.096,158.246
C00767=1030.539,82.471,401.930,168.610,44.094,158.246
C00768=1030.545,82.720,401.911,168.612,44.092,158.246
C00769=1030.551,82.969,401.893,168.615,44.091,158.246
C00770=1030.557,83.219,401.875,168.617,44.089,158.246
C00771=1030.564,83.468,401.856,168.619,44.087,158.246
C00772=1030.569,83.717,401.838,168.622,44.085,158.246
C00773=1030.575,83.966,401.819,168.625,44.083,158.246
C00774=1030.582,84.215,401.800,168.626,44.081,158.245
C00775=1030.588,84.464,401.782,168.629,44.080,158.245
C00776=1030.594,84.714,401.764,168.631,44.078,158.245
C00777=1030.601,84.963,401.745,168.634,44.076,158.245
C00778=1030.607,85.212,401.727,168.637,44.074,158.245
C00779=1030.613,85.461,401.708,168.638,44.072,158.245
C00780=1030.619,85.710,401.690,168.641,44.071,158.245
C00781=1030.625,85.960,401.671,168.644,44.069,158.245
C00782=1030.631,86.209,401.653,168.646,44.067,158.244
C00783=1030.637,86.458,401.634,168.648,44.065,158.244
C00784=1030.644,86.708,401.616,168.650,44.063,158.244
C00785=1030.650,86.957,401.597,168.653,44.062,158.244
C00786=1030.656,87.206,401.579,168.656,44.060,158.244
C00787=1030.663,87.455,401.560,168.657,44.058,158.244
C00788=1030.668,87.705,401.541,168.660,44.056,158.244
C00789=1030.675,87.954,401.523,168.662,44.054,158.243
C00790=1030.680,88.203,401.505,168.665,44.052,158.243
C00791=1030.687,88.452,401.486,168.668,44.050,158.243
C00792=1030.693,88.701,401.467,168.669,44.049,158.243
C00793=1030.700,88.950,401.449,168.672,44.047,158.243
C00794=1030.706,89.200,401.431,168.674,44.045,158.243
C00795=1030.712,89.449,401.412,168.677,44.043,158.243
C00796=1030.718,89.699,401.393,168.680,44.041,158.242
C00797=1030.724,89.948,401.374,168.681,44.040,158.242
C00798=1030.731,90.197,401.355,168.684,44.038,158.242
C00799=1030.737,90.446,401.336,168.687,44.036,158.242
C00800=1030.743,90.695,401.318,168.688,44.034,158.242
C00801=1030.749,90.945,401.298,168.691,44.033,158.242
C00802=1030.755,91.194,401.280,168.694,44.031,158.242
C00803=1030.761,91.443,401.260,168.696,44.029,158.242
C00804=1030.767,91.692,401.242,168.698,44.028,158.241
C00805=1030.774,91.978,401.221,168.701,44.026,158.241
C00806=1030.781,92.263,401.199,168.704,44.024,158.241
C00807=1030.788,92.548,401.177,168.707,44.022,158.241
C00808=1030.795,92.833,401.156,168.709,44.020,158.241
C00809=1030.800,93.083,401.137,168.712,44.018,158.241
C00810=1030.807,93.332,401.118,168.713,44.016,158.241
C00811=1030.812,93.581,401.099,168.716,44.014,158.240
C00812=1030.819,93.830,401.080,168.719,44.013,158.240
C00813=1030.825,94.080,401.061,168.721,44.011,158.240
C00814=1030.831,94.328,401.042,168.724,44.009,158.240
C00815=1030.838,94.578,401.023,168.726,44.008,158.240
C00816=1030.843,94.827,401.004,168.728,44.006,158.240
C00817=1030.850,95.076,400.985,168.731,44.004,158.240
C00818=1030.856,95.326,400.966,168.733,44.002,158.240
C00819=1030.862,95.575,400.947,168.735,44.000,158.239
C00820=1030.868,95.824,400.928,168.738,43.998,158.239
C00821=1030.874,96.073,400.909,168.740,43.996,158.239
C00822=1030.880,96.322,400.891,168.743,43.995,158.239
C00823=1030.886,96.572,400.871,168.745,43.994,158.239
C00824=1030.893,96.820,400.852,168.747,43.992,158.239
C00825=1030.899,97.070,400.833,168.750,43.990,158.239
C00826=1030.905,97.319,400.814,168.752,43.988,158.239
C00827=1030.911,97.568,400.795,168.755,43.986,158.238
C00828=1030.917,97.817,400.776,168.757,43.984,158.238
C00829=1030.923,98.067,400.757,168.759,43.982,158.238
C00830=1030.930,98.316,400.737,168.762,43.981,158.238
C00831=1030.937,98.565,400.719,168.765,43.979,158.238
C00832=1030.942,98.815,400.699,168.767,43.977,158.238
C00833=1030.949,99.064,400.681,168.769,43.976,158.238
C00834=1030.954,99.313,400.661,168.771,43.974,158.237
C00835=1030.961,99.562,400.642,168.774,43.972,158.237
C00836=1030.967,99.811,400.623,168.777,43.970,158.237
C00837=1030.973,100.060,400.604,168.778,43.968,158.237
C00838=1030.979,100.310,400.585,168.781,43.967,158.237
C00839=1030.985,100.558,400.565,168.784,43.965,158.237
C00840=1030.991,100.808,400.546,168.786,43.963,158.237
C00841=1030.998,101.058,400.527,168.788,43.962,158.237
C00842=1031.004,101.306,400.507,168.791,43.960,158.237
C00843=1031.009,101.556,400.487,168.793,43.958,158.236
C00844=1031.016,101.805,400.469,168.796,43.957,158.236
C00845=1031.022,102.054,400.449,168.797,43.955,158.236
C00846=1031.027,102.303,400.430,168.800,43.954,158.236
C00847=1031.033,102.552,400.410,168.803,43.952,158.236
C00848=1031.040,102.801,400.391,168.805,43.950,158.236
C00849=1031.046,103.051,400.372,168.808,43.948,158.236
C00850=1031.052,103.299,400.352,168.810,43.946,158.236
C00851=1031.057,103.549,400.333,168.812,43.945,158.236
C00852=1031.064,103.797,400.313,168.815,43.943,158.235
C00853=1031.070,104.048,400.294,168.818,43.941,158.235
C00854=1031.076,104.297,400.274,168.819,43.940,158.235
C00855=1031.082,104.546,400.254,168.822,43.938,158.235
C00856=1031.088,104.795,400.236,168.825,43.936,158.235
C00857=1031.094,105.044,400.216,168.827,43.935,158.235
C00858=1031.100,105.293,400.197,168.830,43.933,158.235
C00859=1031.106,105.542,400.177,168.831,43.931,158.234
C00860=1031.113,105.792,400.158,168.834,43.930,158.234
C00861=1031.119,106.041,400.138,168.837,43.928,158.234
C00862=1031.125,106.290,400.118,168.839,43.926,158.234
C00863=1031.131,106.539,400.098,168.841,43.924,158.234
C00864=1031.137,106.788,400.080,168.844,43.922,158.234
C00865=1031.143,107.037,400.060,168.846,43.921,158.234
C00866=1031.149,107.287,400.040,168.849,43.919,158.234
C00867=1031.155,107.536,400.020,168.852,43.917,158.234
C00868=1031.162,107.785,400.002,168.853,43.916,158.233
C00869=1031.169,108.070,399.980,168.857,43.914,158.233
C00870=1031.176,108.355,399.956,168.859,43.912,158.233
C00871=1031.183,108.640,399.934,168.862,43.910,158.233
C00872=1031.190,108.926,399.912,168.865,43.908,158.233
C00873=1031.196,109.175,399.892,168.867,43.906,158.233
C00874=1031.202,109.424,399.872,168.870,43.904,158.233
C00875=1031.209,109.673,399.853,168.872,43.902,158.232
C00876=1031.215,109.923,399.833,168.875,43.900,158.232
C00877=1031.221,110.172,399.813,168.877,43.899,158.232
C00878=1031.227,110.420,399.794,168.879,43.897,158.232
C00879=1031.233,110.671,399.774,168.882,43.896,158.232
C00880=1031.239,110.919,399.754,168.885,43.894,158.232
C00881=1031.245,111.168,399.734,168.887,43.892,158.232
C00882=1031.251,111.418,399.715,168.889,43.891,158.232
C00883=1031.257,111.666,399.695,168.892,43.889,158.231
C00884=1031.264,111.916,399.675,168.894,43.887,158.231
C00885=1031.270,112.165,399.656,168.897,43.885,158.231
C00886=1031.276,112.414,399.636,168.900,43.884,158.231
C00887=1031.282,112.663,399.616,168.901,43.882,158.231
C00888=1031.288,112.913,399.596,168.904,43.880,158.231
C00889=1031.294,113.162,399.576,168.907,43.879,158.231
C00890=1031.300,113.410,399.556,168.909,43.877,158.231
C00891=1031.305,113.660,399.536,168.912,43.875,158.231
C00892=1031.312,113.909,399.515,168.914,43.874,158.231
C00893=1031.318,114.158,399.496,168.916,43.872,158.230
C00894=1031.323,114.407,399.476,168.919,43.870,158.230
C00895=1031.329,114.656,399.456,168.922,43.869,158.230
C00896=1031.335,114.906,399.435,168.923,43.868,158.230
C00897=1031.341,115.155,399.415,168.926,43.866,158.230
C00898=1031.347,115.404,399.395,168.929,43.864,158.230
C00899=1031.353,115.652,399.376,168.931,43.863,158.230
C00900=1031.359,115.902,399.355,168.933,43.862,158.230
C00901=1031.365,116.151,399.335,168.936,43.860,158.230
C00902=1031.371,116.400,399.315,168.938,43.858,158.229
C00903=1031.377,116.649,399.295,168.941,43.857,158.229
C00904=1031.383,116.899,399.275,168.944,43.855,158.229
C00905=1031.389,117.148,399.255,168.945,43.853,158.229
C00906=1031.395,117.397,399.235,168.948,43.852,158.229
C00907=1031.401,117.646,399.215,168.951,43.850,158.229
C00908=1031.407,117.895,399.194,168.954,43.849,158.229
C00909=1031.413,118.144,399.174,168.956,43.847,158.229
C00910=1031.418,118.393,399.154,168.958,43.845,158.229
C00911=1031.425,118.643,399.133,168.961,43.844,158.229
C00912=1031.431,118.891,399.114,168.963,43.842,158.229
C00913=1031.437,119.140,399.094,168.966,43.840,158.228
C00914=1031.443,119.390,399.073,168.969,43.839,158.228
C00915=1031.449,119.639,399.053,168.970,43.837,158.228
C00916=1031.455,119.888,399.033,168.973,43.835,158.228
C00917=1031.462,120.137,399.012,168.976,43.834,158.228
C00918=1031.468,120.386,398.992,168.978,43.832,158.228
C00919=1031.473,120.635,398.972,168.981,43.830,158.228
C00920=1031.479,120.885,398.952,168.984,43.829,158.228
C00921=1031.485,121.133,398.932,168.985,43.827,158.228
C00922=1031.491,121.382,398.912,168.988,43.826,158.227
C00923=1031.497,121.632,398.891,168.991,43.824,158.227
C00924=1031.503,121.880,398.870,168.993,43.822,158.227
C00925=1031.510,122.130,398.850,168.996,43.821,158.227
C00926=1031.516,122.379,398.830,168.999,43.819,158.227
C00927=1031.521,122.628,398.809,169.000,43.818,158.227
C00928=1031.528,122.877,398.789,169.003,43.816,158.227
C00929=1031.534,123.126,398.769,169.006,43.814,158.227
C00930=1031.541,123.376,398.749,169.008,43.813,158.227
C00931=1031.546,123.625,398.728,169.011,43.811,158.226
C00932=1031.552,123.873,398.708,169.014,43.809,158.226
C00933=1031.559,124.159,398.684,169.016,43.807,158.226
C00934=1031.567,124.444,398.661,169.019,43.805,158.226
C00935=1031.573,124.729,398.638,169.022,43.804,158.226
C00936=1031.580,125.014,398.614,169.025,43.802,158.226
C00937=1031.587,125.264,398.594,169.028,43.800,158.226
C00938=1031.593,125.512,398.574,169.029,43.798,158.226
C00939=1031.598,125.761,398.553,169.032,43.796,158.225
C00940=1031.605,126.010,398.533,169.035,43.795,158.225
C00941=1031.611,126.259,398.513,169.037,43.793,158.225
C00942=1031.617,126.509,398.492,169.040,43.791,158.225
C00943=1031.623,126.758,398.472,169.043,43.790,158.225
C00944=1031.629,127.007,398.451,169.045,43.788,158.225
C00945=1031.635,127.255,398.431,169.048,43.787,158.225
C00946=1031.642,127.505,398.410,169.051,43.785,158.225
C00947=1031.647,127.754,398.390,169.053,43.784,158.225
C00948=1031.654,128.003,398.369,169.055,43.782,158.225
C00949=1031.660,128.252,398.349,169.058,43.780,158.224
C00950=1031.667,128.501,398.329,169.061,43.779,158.224
C00951=1031.672,128.750,398.307,169.063,43.777,158.224
C00952=1031.679,128.999,398.287,169.066,43.775,158.224
C00953=1031.685,129.248,398.267,169.068,43.773,158.224
C00954=1031.692,129.498,398.247,169.071,43.772,158.224
C00955=1031.697,129.746,398.225,169.074,43.770,158.224
C00956=1031.704,129.996,398.205,169.076,43.768,158.224
C00957=1031.710,130.245,398.185,169.079,43.767,158.224
C00958=1031.716,130.494,398.163,169.081,43.765,158.223
C00959=1031.722,130.743,398.143,169.083,43.763,158.223
C00960=1031.728,130.992,398.122,169.086,43.762,158.223
C00961=1031.735,131.241,398.102,169.089,43.760,158.223
C00962=1031.740,131.490,398.081,169.092,43.759,158.223
C00963=1031.747,131.739,398.060,169.094,43.757,158.223
C00964=1031.752,131.988,398.039,169.097,43.755,158.223
C00965=1031.758,132.238,398.018,169.100,43.754,158.223
C00966=1031.764,132.486,397.998,169.101,43.752,158.223
C00967=1031.770,132.736,397.976,169.104,43.751,158.223
C00968=1031.776,132.984,397.956,169.107,43.749,158.223
C00969=1031.782,133.234,397.935,169.110,43.748,158.223
C00970=1031.788,133.483,397.914,169.112,43.746,158.222
C00971=1031.795,133.732,397.893,169.115,43.745,158.222
C00972=1031.800,133.980,397.872,169.118,43.743,158.222
C00973=1031.807,134.230,397.851,169.120,43.741,158.222
C00974=1031.812,134.478,397.830,169.122,43.740,158.222
C00975=1031.818,134.728,397.809,169.125,43.738,158.222
C00976=1031.825,134.977,397.788,169.127,43.737,158.222
C00977=1031.830,135.226,397.768,169.130,43.735,158.222
C00978=1031.837,135.475,397.747,169.133,43.734,158.222
C00979=1031.843,135.723,397.725,169.135,43.732,158.222
C00980=1031.849,135.973,397.704,169.138,43.730,158.221
C00981=1031.856,136.222,397.683,169.141,43.729,158.221
C00982=1031.861,136.471,397.663,169.143,43.727,158.221
C00983=1031.867,136.720,397.641,169.146,43.726,158.221
C00984=1031.873,136.969,397.620,169.149,43.724,158.221
C00985=1031.879,137.219,397.600,169.151,43.723,158.221
C00986=1031.885,137.468,397.578,169.153,43.721,158.221
C00987=1031.892,137.716,397.557,169.156,43.720,158.221
C00988=1031.897,137.966,397.536,169.159,43.718,158.221
C00989=1031.903,138.214,397.515,169.161,43.716,158.221
C00990=1031.910,138.463,397.494,169.164,43.715,158.221
C00991=1031.916,138.713,397.473,169.167,43.713,158.221
C00992=1031.921,138.961,397.452,169.170,43.712,158.221
C00993=1031.928,139.211,397.430,169.172,43.710,158.220
C00994=1031.934,139.460,397.409,169.175,43.709,158.220
C00995=1031.940,139.708,397.388,169.178,43.707,158.220
C00996=1031.946,139.958,397.367,169.179,43.706,158.220
C00997=1031.952,140.243,397.342,169.183,43.704,158.220
C00998=1031.960,140.528,397.318,169.186,43.703,158.220
C00999=1031.967,140.813,397.294,169.189,43.701,158.220
C01000=1031.973,141.097,397.269,169.192,43.699,158.220
C01001=1031.979,141.347,397.248,169.195,43.698,158.220
C01002=1031.985,141.596,397.226,169.198,43.696,158.220
C01003=1031.991,141.844,397.205,169.200,43.695,158.220
C01004=1031.998,142.093,397.184,169.203,43.693,158.220
C01005=1032.004,142.343,397.162,169.205,43.692,158.219
C01006=1032.009,142.592,397.142,169.208,43.691,158.219
C01007=1032.015,142.841,397.120,169.210,43.689,158.219
C01008=1032.021,143.090,397.098,169.213,43.687,158.219
C01009=1032.027,143.339,397.077,169.216,43.686,158.219
C01010=1032.034,143.587,397.056,169.219,43.684,158.219
C01011=1032.040,143.837,397.034,169.221,43.683,158.219
C01012=1032.046,144.086,397.013,169.224,43.681,158.219
C01013=1032.052,144.334,396.991,169.227,43.679,158.219
C01014=1032.058,144.584,396.970,169.229,43.678,158.219
C01015=1032.064,144.833,396.948,169.232,43.676,158.219
C01016=1032.070,145.082,396.927,169.235,43.675,158.219
C01017=1032.076,145.330,396.905,169.237,43.673,158.219
C01018=1032.082,145.580,396.884,169.240,43.672,158.219
C01019=1032.089,145.829,396.863,169.243,43.670,158.218
C01020=1032.095,146.078,396.841,169.246,43.669,158.218
C01021=1032.100,146.326,396.820,169.248,43.667,158.218
C01022=1032.107,146.575,396.798,169.251,43.666,158.218
C01023=1032.113,146.825,396.776,169.254,43.665,158.218
C01024=1032.119,147.074,396.755,169.257,43.663,158.218
C01025=1032.124,147.322,396.734,169.259,43.662,158.218
C01026=1032.131,147.572,396.712,169.262,43.660,158.218
C01027=1032.137,147.821,396.690,169.265,43.659,158.218
C01028=1032.143,148.070,396.669,169.268,43.657,158.218
C01029=1032.149,148.319,396.647,169.269,43.656,158.218
C01030=1032.154,148.568,396.625,169.272,43.655,158.218
C01031=1032.160,148.817,396.603,169.275,43.653,158.218
C01032=1032.167,149.066,396.581,169.277,43.651,158.218
C01033=1032.173,149.315,396.560,169.280,43.650,158.218
C01034=1032.178,149.564,396.538,169.283,43.648,158.217
C01035=1032.184,149.813,396.517,169.286,43.647,158.217
C01036=1032.191,150.061,396.494,169.289,43.646,158.217
C01037=1032.197,150.311,396.473,169.291,43.644,158.217
C01038=1032.202,150.559,396.451,169.294,43.643,158.217
C01039=1032.208,150.809,396.429,169.297,43.642,158.217
C01040=1032.214,151.058,396.407,169.299,43.640,158.217
C01041=1032.221,151.306,396.385,169.302,43.639,158.217
C01042=1032.227,151.556,396.363,169.305,43.637,158.217
C01043=1032.233,151.805,396.342,169.308,43.636,158.217
C01044=1032.239,152.053,396.321,169.310,43.634,158.217
C01045=1032.244,152.302,396.298,169.313,43.633,158.217
C01046=1032.251,152.551,396.276,169.316,43.631,158.217
C01047=1032.257,152.801,396.254,169.319,43.630,158.217
C01048=1032.263,153.049,396.232,169.322,43.629,158.217
C01049=1032.269,153.298,396.210,169.324,43.627,158.217
C01050=1032.275,153.548,396.189,169.327,43.626,158.217
C01051=1032.281,153.796,396.166,169.330,43.625,158.217
C01052=1032.287,154.045,396.145,169.332,43.623,158.216
C01053=1032.293,154.294,396.123,169.335,43.622,158.216
C01054=1032.299,154.543,396.101,169.338,43.620,158.216
C01055=1032.305,154.792,396.078,169.341,43.619,158.216
C01056=1032.311,155.041,396.056,169.344,43.617,158.216
C01057=1032.317,155.290,396.034,169.346,43.616,158.216
C01058=1032.322,155.539,396.012,169.349,43.615,158.216
C01059=1032.329,155.787,395.990,169.352,43.613,158.216
C01060=1032.335,156.037,395.968,169.355,43.612,158.216
C01061=1032.342,156.321,395.943,169.358,43.610,158.216
C01062=1032.348,156.606,395.918,169.361,43.609,158.216
C01063=1032.355,156.891,395.892,169.365,43.607,158.216
C01064=1032.363,157.175,395.867,169.367,43.605,158.216
C01065=1032.368,157.424,395.845,169.370,43.604,158.216
C01066=1032.375,157.673,395.822,169.373,43.603,158.216
C01067=1032.381,157.922,395.801,169.376,43.601,158.216
C01068=1032.387,158.171,395.778,169.379,43.600,158.216
C01069=1032.393,158.420,395.756,169.381,43.599,158.216
C01070=1032.399,158.669,395.734,169.385,43.597,158.216
C01071=1032.405,158.918,395.712,169.388,43.595,158.216
C01072=1032.411,159.167,395.689,169.391,43.594,158.216
C01073=1032.417,159.416,395.668,169.393,43.593,158.216
C01074=1032.423,159.665,395.645,169.396,43.592,158.216
C01075=1032.430,159.914,395.622,169.399,43.590,158.215
C01076=1032.435,160.163,395.600,169.402,43.589,158.215
C01077=1032.441,160.412,395.577,169.405,43.588,158.215
C01078=1032.446,160.661,395.554,169.407,43.586,158.215
C01079=1032.453,160.910,395.533,169.410,43.585,158.215
C01080=1032.458,161.158,395.510,169.413,43.584,158.215
C01081=1032.463,161.407,395.487,169.416,43.583,158.215
C01082=1032.470,161.656,395.465,169.419,43.582,158.215
C01083=1032.476,161.905,395.442,169.422,43.580,158.215
C01084=1032.481,162.154,395.420,169.424,43.579,158.215
C01085=1032.487,162.403,395.397,169.427,43.578,158.215
C01086=1032.493,162.652,395.374,169.430,43.577,158.215
C01087=1032.499,162.901,395.351,169.433,43.576,158.215
C01088=1032.505,163.149,395.328,169.436,43.574,158.215
C01089=1032.510,163.399,395.306,169.438,43.573,158.215
C01090=1032.517,163.648,395.284,169.441,43.572,158.215
C01091=1032.522,163.896,395.261,169.444,43.571,158.215
C01092=1032.528,164.145,395.238,169.447,43.570,158.215
C01093=1032.534,164.394,395.215,169.450,43.568,158.215
C01094=1032.540,164.643,395.193,169.453,43.567,158.215
C01095=1032.546,164.892,395.170,169.455,43.566,158.215
C01096=1032.552,165.141,395.147,169.458,43.565,158.215
C01097=1032.557,165.390,395.125,169.461,43.564,158.215
C01098=1032.563,165.639,395.102,169.464,43.562,158.215
C01099=1032.569,165.888,395.079,169.467,43.561,158.215
C01100=1032.575,166.137,395.056,169.471,43.560,158.215
C01101=1032.581,166.385,395.033,169.473,43.559,158.215
C01102=1032.587,166.634,395.010,169.476,43.557,158.215
C01103=1032.593,166.883,394.988,169.479,43.556,158.215
C01104=1032.599,167.132,394.965,169.482,43.554,158.215
C01105=1032.605,167.381,394.942,169.484,43.553,158.215
C01106=1032.610,167.630,394.919,169.487,43.552,158.215
C01107=1032.617,167.878,394.897,169.490,43.551,158.215
C01108=1032.623,168.128,394.874,169.493,43.550,158.215
C01109=1032.629,168.377,394.851,169.496,43.548,158.215
C01110=1032.635,168.626,394.828,169.499,43.547,158.215
C01111=1032.640,168.874,394.805,169.502,43.546,158.215
C01112=1032.647,169.123,394.782,169.505,43.545,158.215
C01113=1032.652,169.372,394.759,169.508,43.543,158.215
C01114=1032.658,169.621,394.736,169.511,43.542,158.215
C01115=1032.664,169.870,394.714,169.514,43.541,158.215
C01116=1032.670,170.118,394.691,169.517,43.540,158.215
C01117=1032.677,170.368,394.668,169.519,43.539,158.215
C01118=1032.683,170.616,394.644,169.522,43.537,158.215
C01119=1032.688,170.865,394.621,169.525,43.536,158.215
C01120=1032.694,171.114,394.598,169.529,43.535,158.215
C01121=1032.701,171.363,394.576,169.532,43.534,158.215
C01122=1032.706,171.611,394.553,169.535,43.532,158.215
C01123=1032.712,171.860,394.530,169.537,43.531,158.215
C01124=1032.718,172.110,394.507,169.540,43.530,158.215
C01125=1032.726,172.394,394.480,169.544,43.529,158.215
C01126=1032.733,172.678,394.455,169.547,43.528,158.215
C01127=1032.739,172.962,394.428,169.551,43.526,158.215
C01128=1032.746,173.246,394.401,169.555,43.525,158.215
C01129=1032.752,173.495,394.378,169.557,43.524,158.215
C01130=1032.758,173.744,394.355,169.560,43.522,158.215
C01131=1032.765,173.993,394.333,169.563,43.521,158.215
C01132=1032.771,174.242,394.309,169.566,43.520,158.215
C01133=1032.776,174.490,394.286,169.570,43.519,158.215
C01134=1032.782,174.739,394.263,169.572,43.517,158.215
C01135=1032.789,174.989,394.240,169.575,43.516,158.215
C01136=1032.795,175.237,394.217,169.578,43.515,158.215
C01137=1032.801,175.486,394.194,169.581,43.514,158.215
C01138=1032.807,175.735,394.171,169.585,43.512,158.215
C01139=1032.813,175.984,394.148,169.588,43.511,158.215
C01140=1032.819,176.233,394.124,169.590,43.510,158.215
C01141=1032.825,176.482,394.101,169.593,43.509,158.215
C01142=1032.832,176.731,394.078,169.596,43.508,158.215
C01143=1032.838,176.979,394.055,169.600,43.506,158.215
C01144=1032.844,177.228,394.032,169.603,43.505,158.215
C01145=1032.849,177.477,394.009,169.606,43.504,158.215
C01146=1032.856,177.726,393.985,169.608,43.503,158.215
C01147=1032.862,177.975,393.962,169.612,43.501,158.215
C01148=1032.868,178.223,393.939,169.615,43.500,158.215
C01149=1032.875,178.472,393.915,169.618,43.499,158.215
C01150=1032.881,178.721,393.892,169.621,43.498,158.215
C01151=1032.887,178.969,393.869,169.625,43.496,158.215
C01152=1032.893,179.219,393.845,169.627,43.495,158.215
C01153=1032.899,179.468,393.822,169.630,43.494,158.215
C01154=1032.906,179.716,393.799,169.633,43.493,158.215
C01155=1032.912,179.966,393.776,169.637,43.491,158.215
C01156=1032.918,180.214,393.752,169.640,43.490,158.215
C01157=1032.924,180.463,393.729,169.643,43.489,158.215
C01158=1032.930,180.712,393.705,169.645,43.488,158.215
C01159=1032.936,180.961,393.682,169.649,43.487,158.215
C01160=1032.943,181.209,393.659,169.652,43.486,158.215
C01161=1032.949,181.458,393.636,169.655,43.485,158.215
C01162=1032.956,181.707,393.612,169.659,43.483,158.215
C01163=1032.961,181.956,393.589,169.662,43.482,158.215
C01164=1032.968,182.204,393.565,169.665,43.481,158.215
C01165=1032.974,182.454,393.542,169.667,43.480,158.215
C01166=1032.980,182.702,393.518,169.671,43.478,158.215
C01167=1032.987,182.951,393.496,169.674,43.477,158.215
C01168=1032.992,183.200,393.472,169.677,43.476,158.215
C01169=1032.999,183.449,393.447,169.680,43.476,158.215
C01170=1033.005,183.697,393.424,169.684,43.474,158.215
C01171=1033.010,183.947,393.400,169.687,43.473,158.215
C01172=1033.017,184.196,393.376,169.690,43.472,158.216
C01173=1033.022,184.444,393.352,169.692,43.471,158.216
C01174=1033.028,184.692,393.328,169.696,43.470,158.216
C01175=1033.034,184.942,393.304,169.699,43.469,158.216
C01176=1033.040,185.191,393.281,169.702,43.468,158.216
C01177=1033.046,185.439,393.257,169.705,43.468,158.216
C01178=1033.051,185.688,393.232,169.709,43.466,158.216
C01179=1033.058,185.936,393.209,169.712,43.466,158.216
C01180=1033.063,186.186,393.184,169.715,43.464,158.216
C01181=1033.069,186.434,393.161,169.718,43.463,158.216
C01182=1033.075,186.683,393.136,169.722,43.463,158.216
C01183=1033.081,186.932,393.112,169.725,43.461,158.216
C01184=1033.087,187.180,393.088,169.728,43.461,158.216
C01185=1033.093,187.430,393.065,169.730,43.460,158.216
C01186=1033.099,187.678,393.041,169.734,43.458,158.216
C01187=1033.105,187.927,393.016,169.737,43.458,158.216
C01188=1033.111,188.176,392.993,169.740,43.456,158.216
C01189=1033.118,188.459,392.965,169.744,43.456,158.217
C01190=1033.125,188.743,392.937,169.748,43.454,158.217
C01191=1033.132,189.027,392.910,169.751,43.453,158.217
C01192=1033.138,189.311,392.882,169.755,43.452,158.217
C01193=1033.144,189.560,392.858,169.758,43.451,158.217
C01194=1033.150,189.809,392.834,169.762,43.451,158.217
C01195=1033.156,190.057,392.810,169.765,43.449,158.217
C01196=1033.162,190.306,392.786,169.767,43.448,158.217
C01197=1033.168,190.554,392.762,169.772,43.447,158.217
C01198=1033.174,190.804,392.737,169.774,43.446,158.217
C01199=1033.180,191.052,392.714,169.777,43.446,158.217
C01200=1033.186,191.301,392.689,169.781,43.444,158.217
C01201=1033.193,191.550,392.665,169.784,43.444,158.217
C01202=1033.198,191.798,392.640,169.787,43.443,158.217
C01203=1033.205,192.047,392.616,169.791,43.442,158.218
C01204=1033.210,192.296,392.592,169.794,43.441,158.218
C01205=1033.217,192.545,392.568,169.797,43.440,158.218
C01206=1033.222,192.793,392.544,169.801,43.439,158.218
C01207=1033.229,193.042,392.520,169.804,43.438,158.218
C01208=1033.235,193.292,392.495,169.807,43.437,158.218
C01209=1033.241,193.539,392.471,169.811,43.436,158.218
C01210=1033.247,193.789,392.446,169.814,43.435,158.218
C01211=1033.253,194.037,392.422,169.817,43.435,158.218
C01212=1033.259,194.286,392.398,169.820,43.433,158.218
C01213=1033.266,194.535,392.374,169.823,43.433,158.218
C01214=1033.271,194.783,392.349,169.827,43.431,158.218
C01215=1033.278,195.032,392.325,169.830,43.431,158.218
C01216=1033.284,195.281,392.300,169.833,43.430,158.218
C01217=1033.290,195.530,392.276,169.837,43.429,158.219
C01218=1033.296,195.778,392.251,169.840,43.428,158.219
C01219=1033.303,196.027,392.227,169.844,43.427,158.219
C01220=1033.308,196.276,392.203,169.847,43.426,158.219
C01221=1033.314,196.525,392.179,169.850,43.425,158.219
C01222=1033.321,196.773,392.153,169.854,43.424,158.219
C01223=1033.327,197.022,392.130,169.857,43.423,158.219
C01224=1033.333,197.271,392.105,169.861,43.422,158.219
C01225=1033.340,197.519,392.080,169.864,43.421,158.219
C01226=1033.345,197.768,392.056,169.868,43.420,158.219
C01227=1033.352,198.017,392.032,169.871,43.420,158.219
C01228=1033.358,198.266,392.007,169.873,43.418,158.219
C01229=1033.364,198.515,391.983,169.878,43.418,158.220
C01230=1033.370,198.763,391.958,169.881,43.417,158.220
C01231=1033.377,199.012,391.934,169.884,43.416,158.220
C01232=1033.383,199.261,391.909,169.887,43.415,158.220
C01233=1033.389,199.509,391.884,169.891,43.414,158.220
C01234=1033.395,199.758,391.860,169.894,43.413,158.220
C01235=1033.402,200.006,391.835,169.898,43.412,158.220
C01236=1033.408,200.255,391.811,169.901,43.411,158.220
C01237=1033.414,200.504,391.785,169.904,43.411,158.220
C01238=1033.420,200.753,391.761,169.908,43.409,158.220
C01239=1033.426,201.001,391.736,169.911,43.409,158.220
C01240=1033.432,201.250,391.712,169.915,43.408,158.221
C01241=1033.438,201.499,391.686,169.918,43.408,158.221
C01242=1033.444,201.748,391.661,169.922,43.406,158.221
C01243=1033.450,201.996,391.637,169.925,43.406,158.221
C01244=1033.456,202.245,391.611,169.929,43.405,158.221
C01245=1033.463,202.493,391.587,169.932,43.404,158.221
C01246=1033.469,202.743,391.562,169.935,43.404,158.221
C01247=1033.475,202.991,391.537,169.939,43.403,158.221
C01248=1033.481,203.239,391.512,169.942,43.402,158.222
C01249=1033.486,203.488,391.487,169.946,43.401,158.222
C01250=1033.493,203.737,391.462,169.949,43.401,158.222
C01251=1033.499,203.986,391.436,169.953,43.400,158.222
C01252=1033.505,204.234,391.411,169.956,43.399,158.222
C01253=1033.531,205.284,391.306,170.290,43.503,158.271
C01254=1033.541,205.629,391.270,170.293,43.503,158.271
C01255=1033.550,205.974,391.233,170.296,43.503,158.271
C01256=1033.559,206.319,391.196,170.299,43.503,158.271
C01257=1033.569,206.664,391.159,170.304,43.503,158.272
C01258=1033.575,206.912,391.133,170.306,43.503,158.272
C01259=1033.582,207.161,391.107,170.308,43.503,158.272
C01260=1033.589,207.409,391.081,170.311,43.503,158.272
C01261=1033.595,207.658,391.054,170.313,43.503,158.273
C01262=1033.602,207.907,391.027,170.316,43.504,158.273
C01263=1033.609,208.155,391.001,170.319,43.503,158.273
C01264=1033.616,208.404,390.975,170.321,43.503,158.273
C01265=1033.622,208.652,390.948,170.323,43.504,158.274
C01266=1033.629,208.901,390.922,170.326,43.503,158.274
C01267=1033.636,209.149,390.895,170.329,43.503,158.274
C01268=1033.643,209.397,390.869,170.331,43.504,158.274
C01269=1033.649,209.646,390.842,170.334,43.504,158.274
C01270=1033.656,209.895,390.815,170.336,43.503,158.274
C01271=1033.663,210.143,390.789,170.338,43.504,158.275
C01272=1033.669,210.392,390.762,170.342,43.504,158.275
C01273=1033.677,210.640,390.735,170.344,43.504,158.275
C01274=1033.683,210.888,390.709,170.346,43.504,158.275
C01275=1033.689,211.137,390.682,170.349,43.504,158.276
C01276=1033.697,211.386,390.655,170.351,43.504,158.276
C01277=1033.702,211.634,390.629,170.354,43.504,158.276
C01278=1033.710,211.883,390.602,170.357,43.504,158.276
C01279=1033.716,212.132,390.575,170.359,43.504,158.276
C01280=1033.723,212.380,390.549,170.362,43.504,158.277
C01281=1033.729,212.628,390.521,170.364,43.504,158.277
C01282=1033.736,212.877,390.494,170.367,43.505,158.277
C01283=1033.742,213.125,390.468,170.370,43.505,158.278
C01284=1033.750,213.373,390.441,170.372,43.504,158.278
C01285=1033.756,213.622,390.414,170.374,43.505,158.278
C01286=1033.763,213.870,390.388,170.377,43.505,158.278
C01287=1033.769,214.119,390.360,170.380,43.505,158.278
C01288=1033.776,214.368,390.333,170.383,43.505,158.279
C01289=1033.782,214.616,390.307,170.385,43.505,158.279
C01290=1033.789,214.864,390.280,170.387,43.505,158.279
C01291=1033.796,215.113,390.253,170.390,43.505,158.279
C01292=1033.803,215.361,390.226,170.393,43.505,158.279
C01293=1033.809,215.610,390.199,170.396,43.505,158.280
C01294=1033.816,215.858,390.172,170.398,43.506,158.280
C01295=1033.823,216.107,390.145,170.400,43.505,158.280
C01296=1033.830,216.356,390.118,170.403,43.505,158.280
C01297=1033.836,216.603,390.091,170.406,43.506,158.281
C01298=1033.843,216.852,390.065,170.409,43.506,158.281
C01299=1033.850,217.101,390.037,170.411,43.506,158.281
C01300=1033.857,217.349,390.010,170.413,43.506,158.281
C01301=1033.863,217.597,389.983,170.416,43.506,158.282
C01302=1033.870,217.846,389.957,170.419,43.506,158.282
C01303=1033.877,218.094,389.929,170.422,43.506,158.282
C01304=1033.884,218.343,389.902,170.424,43.506,158.282
C01305=1033.891,218.591,389.875,170.428,43.506,158.283
C01306=1033.897,218.840,389.849,170.430,43.507,158.283
C01307=1033.904,219.088,389.821,170.433,43.506,158.283
C01308=1033.911,219.337,389.795,170.435,43.506,158.283
C01309=1033.918,219.585,389.767,170.438,43.506,158.283
C01310=1033.926,219.936,389.729,170.442,43.506,158.284
C01311=1033.936,220.287,389.689,170.445,43.507,158.284
C01312=1033.946,220.637,389.651,170.449,43.507,158.284
C01313=1033.955,220.988,389.613,170.453,43.507,158.285
C01314=1033.961,221.236,389.585,170.456,43.507,158.285
C01315=1033.968,221.485,389.558,170.458,43.507,158.285
C01316=1033.974,221.734,389.531,170.461,43.507,158.286
C01317=1033.982,221.982,389.504,170.464,43.508,158.286
C01318=1033.988,222.231,389.476,170.466,43.508,158.286
C01319=1033.995,222.478,389.448,170.469,43.508,158.286
C01320=1034.001,222.727,389.421,170.471,43.508,158.287
C01321=1034.008,222.976,389.394,170.475,43.508,158.287
C01322=1034.015,223.224,389.367,170.477,43.509,158.287
C01323=1034.022,223.472,389.339,170.480,43.509,158.287
C01324=1034.028,223.721,389.312,170.482,43.509,158.288
C01325=1034.035,223.970,389.284,170.486,43.509,158.288
C01326=1034.041,224.218,389.257,170.488,43.509,158.288
C01327=1034.048,224.466,389.230,170.491,43.509,158.288
C01328=1034.055,224.714,389.202,170.493,43.510,158.289
C01329=1034.061,224.963,389.175,170.497,43.510,158.289
C01330=1034.068,225.212,389.147,170.499,43.510,158.289
C01331=1034.075,225.460,389.119,170.502,43.510,158.289
C01332=1034.082,225.708,389.092,170.504,43.510,158.290
C01333=1034.089,225.957,389.065,170.507,43.510,158.290
C01334=1034.095,226.205,389.037,170.510,43.510,158.290
C01335=1034.102,226.454,389.009,170.513,43.510,158.290
C01336=1034.109,226.702,388.981,170.515,43.510,158.291
C01337=1034.115,226.951,388.954,170.518,43.510,158.291
C01338=1034.123,227.199,388.927,170.521,43.511,158.291
C01339=1034.129,227.447,388.900,170.524,43.511,158.291
C01340=1034.135,227.695,388.872,170.526,43.511,158.292
C01341=1034.142,227.944,388.844,170.529,43.511,158.292
C01342=1034.149,228.192,388.817,170.532,43.511,158.292
C01343=1034.155,228.441,388.789,170.535,43.511,158.292
C01344=1034.162,228.689,388.761,170.537,43.512,158.293
C01345=1034.169,228.938,388.733,170.540,43.512,158.293
C01346=1034.175,229.186,388.706,170.543,43.512,158.293
C01347=1034.182,229.434,388.677,170.546,43.513,158.294
C01348=1034.189,229.682,388.650,170.549,43.513,158.294
C01349=1034.196,229.931,388.622,170.552,43.513,158.294
C01350=1034.202,230.179,388.594,170.555,43.513,158.294
C01351=1034.209,230.428,388.566,170.557,43.513,158.295
C01352=1034.216,230.676,388.539,170.560,43.514,158.295
C01353=1034.223,230.924,388.511,170.563,43.514,158.295
C01354=1034.228,231.173,388.483,170.566,43.514,158.295
C01355=1034.235,231.422,388.455,170.568,43.514,158.296
C01356=1034.242,231.670,388.426,170.571,43.514,158.296
C01357=1034.249,231.918,388.399,170.574,43.514,158.296
C01358=1034.255,232.166,388.371,170.577,43.515,158.297
C01359=1034.262,232.415,388.343,170.579,43.515,158.297
C01360=1034.268,232.663,388.314,170.583,43.515,158.297
C01361=1034.275,232.911,388.286,170.586,43.516,158.297
C01362=1034.282,233.160,388.259,170.588,43.516,158.298
C01363=1034.288,233.408,388.231,170.591,43.516,158.298
C01364=1034.295,233.656,388.203,170.594,43.516,158.298
C01365=1034.301,233.905,388.174,170.597,43.517,158.299
C01366=1034.311,234.248,388.136,170.600,43.517,158.299
C01367=1034.320,234.591,388.097,170.605,43.517,158.299
C01368=1034.329,234.934,388.058,170.608,43.518,158.300
C01369=1034.339,235.277,388.019,170.613,43.518,158.300
C01370=1034.345,235.526,387.991,170.616,43.518,158.300
C01371=1034.352,235.774,387.963,170.618,43.518,158.301
C01372=1034.359,236.023,387.934,170.622,43.519,158.301
C01373=1034.365,236.272,387.907,170.624,43.519,158.301
C01374=1034.372,236.519,387.878,170.627,43.519,158.302
C01375=1034.378,236.768,387.850,170.630,43.519,158.302
C01376=1034.385,237.016,387.821,170.633,43.520,158.302
C01377=1034.392,237.264,387.794,170.636,43.520,158.302
C01378=1034.399,237.513,387.766,170.638,43.521,158.303
C01379=1034.405,237.761,387.737,170.642,43.521,158.303
C01380=1034.412,238.009,387.709,170.645,43.521,158.303
C01381=1034.419,238.258,387.680,170.647,43.521,158.304
C01382=1034.426,238.506,387.653,170.650,43.521,158.304
C01383=1034.432,238.755,387.624,170.654,43.522,158.304
C01384=1034.439,239.003,387.596,170.656,43.522,158.305
C01385=1034.446,239.251,387.568,170.659,43.522,158.305
C01386=1034.452,239.500,387.539,170.662,43.522,158.305
C01387=1034.459,239.748,387.510,170.665,43.522,158.305
C01388=1034.466,239.996,387.482,170.668,43.523,158.306
C01389=1034.472,240.245,387.454,170.670,43.523,158.306
C01390=1034.479,240.492,387.425,170.674,43.524,158.306
C01391=1034.486,240.741,387.397,170.677,43.524,158.307
C01392=1034.492,240.989,387.368,170.679,43.524,158.307
C01393=1034.499,241.237,387.340,170.683,43.525,158.307
C01394=1034.506,241.486,387.311,170.686,43.525,158.308
C01395=1034.513,241.734,387.283,170.688,43.525,158.308
C01396=1034.519,241.982,387.254,170.692,43.526,158.308
C01397=1034.525,242.230,387.225,170.694,43.526,158.308
C01398=1034.532,242.479,387.197,170.697,43.527,158.309
C01399=1034.539,242.728,387.168,170.701,43.527,158.309
C01400=1034.546,242.975,387.139,170.703,43.527,158.309
C01401=1034.552,243.224,387.110,170.706,43.528,158.310
C01402=1034.559,243.472,387.082,170.710,43.528,158.310
C01403=1034.565,243.720,387.053,170.712,43.528,158.310
C01404=1034.573,243.969,387.025,170.715,43.529,158.311
C01405=1034.579,244.217,386.995,170.719,43.529,158.311
C01406=1034.586,244.465,386.968,170.721,43.529,158.311
C01407=1034.592,244.713,386.939,170.724,43.530,158.312
C01408=1034.598,244.962,386.910,170.728,43.530,158.312
C01409=1034.605,245.210,386.880,170.730,43.531,158.312
C01410=1034.612,245.458,386.852,170.733,43.531,158.313
C01411=1034.618,245.706,386.823,170.737,43.531,158.313
C01412=1034.624,245.954,386.794,170.739,43.532,158.313
C01413=1034.631,246.203,386.765,170.743,43.532,158.314
C01414=1034.637,246.451,386.735,170.746,43.532,158.314
C01415=1034.644,246.699,386.707,170.748,43.533,158.315
C01416=1034.651,246.947,386.678,170.752,43.533,158.315
C01417=1034.657,247.196,386.649,170.755,43.533,158.315
C01418=1034.664,247.444,386.619,170.757,43.534,158.315
C01419=1034.670,247.692,386.590,170.761,43.534,158.316
C01420=1034.676,247.941,386.561,170.764,43.535,158.316
C01421=1034.683,248.188,386.533,170.766,43.535,158.316
C01422=1034.692,248.526,386.493,170.771,43.536,158.317
C01423=1034.701,248.863,386.453,170.775,43.536,158.317
C01424=1034.710,249.201,386.414,170.779,43.538,158.318
C01425=1034.719,249.538,386.374,170.783,43.538,158.318
C01426=1034.726,249.786,386.345,170.787,43.538,158.319
C01427=1034.732,250.035,386.316,170.790,43.539,158.319
C01428=1034.738,250.283,386.287,170.792,43.539,158.319
C01429=1034.746,250.531,386.258,170.796,43.540,158.320
C01430=1034.752,250.779,386.229,170.799,43.540,158.320
C01431=1034.759,251.028,386.200,170.802,43.541,158.321
C01432=1034.766,251.276,386.170,170.805,43.541,158.321
C01433=1034.772,251.524,386.140,170.808,43.541,158.321
C01434=1034.778,251.772,386.111,170.812,43.542,158.322
C01435=1034.786,252.021,386.083,170.814,43.542,158.322
C01436=1034.792,252.268,386.053,170.817,43.542,158.322
C01437=1034.799,252.517,386.023,170.821,43.543,158.323
C01438=1034.805,252.765,385.994,170.824,43.543,158.323
C01439=1034.812,253.013,385.965,170.827,43.544,158.323
C01440=1034.819,253.261,385.935,170.830,43.544,158.324
C01441=1034.825,253.509,385.906,170.833,43.545,158.324
C01442=1034.833,253.758,385.877,170.837,43.545,158.324
C01443=1034.839,254.006,385.848,170.840,43.546,158.325
C01444=1034.846,254.254,385.818,170.842,43.546,158.325
C01445=1034.852,254.502,385.789,170.846,43.547,158.325
C01446=1034.859,254.751,385.760,170.849,43.547,158.326
C01447=1034.866,254.999,385.730,170.852,43.547,158.326
C01448=1034.872,255.247,385.701,170.856,43.548,158.327
C01449=1034.880,255.495,385.671,170.858,43.548,158.327
C01450=1034.886,255.743,385.642,170.862,43.549,158.327
C01451=1034.893,255.992,385.613,170.865,43.549,158.328
C01452=1034.900,256.239,385.583,170.868,43.550,158.328
C01453=1034.906,256.488,385.554,170.872,43.550,158.328
C01454=1034.913,256.736,385.524,170.874,43.551,158.329
C01455=1034.920,256.985,385.495,170.878,43.551,158.329
C01456=1034.927,257.232,385.466,170.881,43.551,158.329
C01457=1034.934,257.481,385.436,170.884,43.552,158.330
C01458=1034.940,257.729,385.407,170.888,43.552,158.330
C01459=1034.947,257.977,385.377,170.891,43.553,158.331
C01460=1034.954,258.225,385.348,170.894,43.554,158.331
C01461=1034.961,258.473,385.318,170.897,43.554,158.331
C01462=1034.968,258.722,385.288,170.900,43.554,158.332
C01463=1034.974,258.970,385.259,170.904,43.554,158.332
C01464=1034.981,259.218,385.229,170.907,43.555,158.332
C01465=1034.988,259.466,385.200,170.910,43.556,158.333
C01466=1034.995,259.714,385.170,170.914,43.556,158.333
C01467=1035.002,259.962,385.141,170.916,43.557,158.333
C01468=1035.009,260.210,385.111,170.919,43.557,158.334
C01469=1035.016,260.459,385.081,170.923,43.558,158.334
C01470=1035.022,260.707,385.052,170.926,43.558,158.335
C01471=1035.029,260.955,385.022,170.930,43.558,158.335
C01472=1035.036,261.203,384.992,170.933,43.559,158.335
C01473=1035.044,261.451,384.963,170.937,43.560,158.336
C01474=1035.050,261.699,384.932,170.940,43.560,158.336
C01475=1035.056,261.947,384.903,170.943,43.560,158.336
C01476=1035.063,262.196,384.873,170.946,43.561,158.337
C01477=1035.070,262.443,384.843,170.949,43.562,158.337
C01478=1035.079,262.780,384.802,170.954,43.562,158.338
C01479=1035.087,263.115,384.762,170.959,43.564,158.338
C01480=1035.097,263.452,384.721,170.963,43.564,158.339
C01481=1035.106,263.788,384.680,170.968,43.565,158.339
C01482=1035.113,264.036,384.650,170.971,43.565,158.340
C01483=1035.119,264.283,384.620,170.974,43.566,158.340
C01484=1035.126,264.532,384.590,170.977,43.567,158.341
C01485=1035.133,264.780,384.560,170.980,43.567,158.341
C01486=1035.139,265.027,384.530,170.984,43.568,158.342
C01487=1035.147,265.276,384.500,170.987,43.568,158.342
C01488=1035.153,265.524,384.469,170.991,43.569,158.342
C01489=1035.160,265.772,384.439,170.994,43.570,158.343
C01490=1035.167,266.020,384.409,170.998,43.570,158.343
C01491=1035.173,266.268,384.378,171.001,43.571,158.344
C01492=1035.180,266.516,384.349,171.005,43.572,158.344
C01493=1035.187,266.764,384.319,171.008,43.572,158.344
C01494=1035.193,267.013,384.288,171.011,43.573,158.345
C01495=1035.200,267.260,384.258,171.014,43.573,158.345
C01496=1035.207,267.508,384.228,171.017,43.574,158.346
C01497=1035.213,267.757,384.197,171.021,43.575,158.346
C01498=1035.221,268.005,384.167,171.024,43.575,158.346
C01499=1035.226,268.253,384.137,171.028,43.576,158.347
C01500=1035.234,268.501,384.107,171.031,43.577,158.347
C01501=1035.241,268.749,384.076,171.035,43.577,158.348
C01502=1035.247,268.997,384.045,171.038,43.578,158.348
C01503=1035.254,269.245,384.015,171.042,43.579,158.349
C01504=1035.260,269.493,383.985,171.045,43.579,158.349
C01505=1035.268,269.742,383.955,171.049,43.580,158.349
C01506=1035.274,269.989,383.923,171.052,43.581,158.350
C01507=1035.281,270.237,383.893,171.056,43.581,158.350
C01508=1035.287,270.486,383.863,171.059,43.582,158.351
C01509=1035.294,270.734,383.832,171.062,43.583,158.351
C01510=1035.301,270.981,383.801,171.066,43.583,158.352
C01511=1035.308,271.229,383.771,171.069,43.584,158.352
C01512=1035.314,271.478,383.741,171.072,43.585,158.352
C01513=1035.322,271.725,383.710,171.075,43.586,158.353
C01514=1035.328,271.974,383.679,171.079,43.586,158.353
C01515=1035.334,272.222,383.649,171.082,43.587,158.354
C01516=1035.341,272.469,383.618,171.086,43.588,158.354
C01517=1035.348,272.718,383.587,171.089,43.588,158.355
C01518=1035.355,272.965,383.556,171.093,43.589,158.355
C01519=1035.362,273.214,383.526,171.096,43.590,158.356
C01520=1035.367,273.462,383.495,171.100,43.591,158.356
C01521=1035.375,273.709,383.464,171.103,43.592,158.357
C01522=1035.381,273.958,383.434,171.107,43.592,158.357
C01523=1035.389,274.205,383.403,171.110,43.593,158.357
C01524=1035.395,274.454,383.372,171.114,43.594,158.358
C01525=1035.402,274.702,383.341,171.117,43.594,158.358
C01526=1035.408,274.950,383.310,171.121,43.595,158.359
C01527=1035.415,275.197,383.279,171.124,43.596,158.359
C01528=1035.422,275.445,383.248,171.128,43.597,158.360
C01529=1035.428,275.694,383.217,171.132,43.598,158.360
C01530=1035.436,275.941,383.186,171.135,43.598,158.361
C01531=1035.442,276.190,383.156,171.139,43.599,158.361
C01532=1035.449,276.438,383.124,171.142,43.600,158.362
C01533=1035.456,276.685,383.094,171.145,43.600,158.362
C01534=1035.465,277.026,383.052,171.151,43.601,158.363
C01535=1035.475,277.366,383.009,171.156,43.602,158.363
C01536=1035.484,277.707,382.967,171.161,43.603,158.364
C01537=1035.493,278.048,382.924,171.165,43.605,158.365
C01538=1035.500,278.295,382.892,171.169,43.606,158.365
C01539=1035.506,278.544,382.861,171.173,43.606,158.366
C01540=1035.513,278.792,382.830,171.176,43.607,158.366
C01541=1035.520,279.040,382.799,171.180,43.608,158.367
C01542=1035.527,279.288,382.767,171.183,43.609,158.367
C01543=1035.533,279.536,382.736,171.187,43.610,158.367
C01544=1035.540,279.784,382.704,171.190,43.611,158.368
C01545=1035.547,280.031,382.673,171.195,43.612,158.369
C01546=1035.553,280.279,382.643,171.198,43.612,158.369
C01547=1035.559,280.527,382.611,171.202,43.614,158.370
C01548=1035.566,280.775,382.580,171.206,43.614,158.370
C01549=1035.573,281.023,382.548,171.209,43.615,158.370
C01550=1035.580,281.271,382.517,171.213,43.616,158.371
C01551=1035.587,281.518,382.486,171.216,43.617,158.371
C01552=1035.594,281.766,382.455,171.220,43.617,158.372
C01553=1035.600,282.014,382.423,171.223,43.619,158.373
C01554=1035.607,282.262,382.392,171.227,43.619,158.373
C01555=1035.614,282.510,382.360,171.231,43.621,158.374
C01556=1035.621,282.758,382.329,171.234,43.621,158.374
C01557=1035.628,283.007,382.297,171.239,43.622,158.374
C01558=1035.635,283.254,382.266,171.242,43.623,158.375
C01559=1035.641,283.502,382.234,171.246,43.624,158.375
C01560=1035.648,283.750,382.203,171.250,43.625,158.376
C01561=1035.655,283.998,382.171,171.253,43.626,158.377
C01562=1035.661,284.246,382.140,171.256,43.626,158.377
C01563=1035.669,284.493,382.108,171.260,43.628,158.378
C01564=1035.675,284.741,382.076,171.264,43.628,158.378
C01565=1035.682,284.989,382.045,171.268,43.629,158.379
C01566=1035.689,285.237,382.013,171.272,43.630,158.379
C01567=1035.695,285.485,381.982,171.276,43.631,158.380
C01568=1035.703,285.734,381.950,171.279,43.632,158.380
C01569=1035.709,285.981,381.919,171.283,43.633,158.381
C01570=1035.716,286.229,381.887,171.286,43.634,158.381
C01571=1035.723,286.477,381.855,171.291,43.634,158.382
C01572=1035.730,286.725,381.824,171.294,43.636,158.382
C01573=1035.737,286.972,381.792,171.298,43.637,158.383
C01574=1035.744,287.220,381.760,171.302,43.638,158.383
C01575=1035.750,287.468,381.728,171.305,43.639,158.384
C01576=1035.757,287.717,381.696,171.309,43.640,158.384
C01577=1035.764,287.964,381.664,171.314,43.641,158.385
C01578=1035.771,288.212,381.633,171.317,43.641,158.385
C01579=1035.778,288.459,381.601,171.321,43.643,158.386
C01580=1035.785,288.707,381.569,171.324,43.644,158.387
C01581=1035.791,288.956,381.537,171.328,43.645,158.387
C01582=1035.798,289.203,381.505,171.332,43.646,158.388
C01583=1035.805,289.451,381.473,171.336,43.647,158.388
C01584=1035.812,289.698,381.441,171.340,43.648,158.389
C01585=1035.818,289.947,381.409,171.344,43.649,158.389
C01586=1035.825,290.194,381.377,171.347,43.650,158.390
C01587=1035.832,290.442,381.345,171.351,43.651,158.390
C01588=1035.839,290.690,381.313,171.355,43.652,158.391
C01589=1035.845,290.938,381.281,171.359,43.653,158.391
C01590=1035.856,291.290,381.235,171.364,43.654,158.392
C01591=1035.865,291.643,381.190,171.370,43.656,158.393
C01592=1035.875,291.996,381.143,171.376,43.657,158.394
C01593=1035.884,292.348,381.098,171.381,43.659,158.395
C01594=1035.892,292.596,381.066,171.384,43.660,158.395
C01595=1035.898,292.843,381.033,171.389,43.661,158.396
C01596=1035.905,293.091,381.001,171.393,43.662,158.396
C01597=1035.913,293.339,380.969,171.396,43.663,158.397
C01598=1035.919,293.587,380.936,171.400,43.665,158.397
C01599=1035.926,293.835,380.905,171.405,43.666,158.398
C01600=1035.933,294.083,380.872,171.408,43.666,158.399
C01601=1035.940,294.330,380.839,171.412,43.668,158.399
C01602=1035.947,294.578,380.807,171.416,43.669,158.400
C01603=1035.953,294.826,380.774,171.420,43.670,158.400
C01604=1035.960,295.074,380.743,171.424,43.671,158.401
C01605=1035.967,295.322,380.710,171.428,43.672,158.402
C01606=1035.973,295.569,380.677,171.432,43.674,158.402
C01607=1035.980,295.817,380.645,171.436,43.675,158.403
C01608=1035.987,296.065,380.612,171.440,43.676,158.403
C01609=1035.993,296.312,380.579,171.444,43.677,158.404
C01610=1036.000,296.561,380.546,171.447,43.679,158.405
C01611=1036.007,296.808,380.514,171.452,43.680,158.405
C01612=1036.013,297.055,380.481,171.456,43.681,158.406
C01613=1036.020,297.304,380.448,171.460,43.682,158.406
C01614=1036.026,297.551,380.415,171.463,43.684,158.407
C01615=1036.034,297.798,380.383,171.468,43.685,158.408
C01616=1036.041,298.046,380.349,171.472,43.686,158.408
C01617=1036.047,298.294,380.317,171.475,43.687,158.409
C01618=1036.053,298.541,380.284,171.480,43.688,158.409
C01619=1036.061,298.789,380.251,171.484,43.689,158.410
C01620=1036.067,299.037,380.219,171.488,43.691,158.411
C01621=1036.074,299.285,380.186,171.491,43.692,158.411
C01622=1036.081,299.532,380.152,171.496,43.693,158.412
C01623=1036.088,299.780,380.120,171.500,43.694,158.413
C01624=1036.095,300.028,380.087,171.504,43.696,158.413
C01625=1036.101,300.276,380.054,171.508,43.697,158.414
C01626=1036.108,300.524,380.021,171.512,43.699,158.415
C01627=1036.115,300.770,379.988,171.516,43.700,158.415
C01628=1036.122,301.019,379.955,171.521,43.701,158.416
C01629=1036.128,301.266,379.922,171.524,43.702,158.416
C01630=1036.135,301.514,379.889,171.528,43.703,158.417
C01631=1036.143,301.761,379.856,171.533,43.704,158.418
C01632=1036.149,302.010,379.823,171.536,43.706,158.418
C01633=1036.156,302.257,379.790,171.541,43.707,158.419
C01634=1036.163,302.505,379.757,171.545,43.709,158.420
C01635=1036.169,302.752,379.724,171.549,43.710,158.420
C01636=1036.177,303.000,379.691,171.554,43.711,158.421
C01637=1036.184,303.248,379.658,171.557,43.712,158.421
C01638=1036.191,303.495,379.624,171.561,43.714,158.422
C01639=1036.198,303.743,379.591,171.566,43.715,158.423
C01640=1036.205,303.991,379.559,171.570,43.716,158.423
C01641=1036.212,304.238,379.525,171.574,43.718,158.424
C01642=1036.218,304.486,379.492,171.578,43.719,158.425
C01643=1036.225,304.734,379.459,171.582,43.721,158.425
C01644=1036.232,304.982,379.425,171.587,43.722,158.426
C01645=1036.239,305.229,379.393,171.591,43.723,158.427
C01646=1036.250,305.599,379.342,171.597,43.725,158.428
C01647=1036.260,305.967,379.293,171.604,43.727,158.429
C01648=1036.270,306.337,379.243,171.610,43.729,158.430
C01649=1036.281,306.706,379.193,171.616,43.731,158.431
C01650=1036.288,306.955,379.160,171.620,43.732,158.431
C01651=1036.295,307.202,379.127,171.625,43.733,158.432
C01652=1036.303,307.449,379.094,171.629,43.735,158.433
C01653=1036.310,307.697,379.061,171.633,43.736,158.433
C01654=1036.316,307.944,379.027,171.637,43.738,158.434
C01655=1036.324,308.192,378.993,171.642,43.739,158.435
C01656=1036.330,308.440,378.960,171.646,43.741,158.435
C01657=1036.338,308.688,378.926,171.651,43.742,158.436
C01658=1036.345,308.935,378.894,171.654,43.743,158.437
C01659=1036.352,309.182,378.860,171.659,43.745,158.437
C01660=1036.359,309.430,378.826,171.663,43.746,158.438
C01661=1036.366,309.678,378.793,171.668,43.747,158.439
C01662=1036.374,309.926,378.759,171.672,43.749,158.439
C01663=1036.381,310.173,378.726,171.677,43.750,158.440
C01664=1036.388,310.420,378.692,171.680,43.752,158.441
C01665=1036.395,310.668,378.658,171.685,43.753,158.442
C01666=1036.402,310.916,378.625,171.689,43.755,158.442
C01667=1036.409,311.164,378.591,171.694,43.756,158.443
C01668=1036.417,311.412,378.558,171.698,43.757,158.444
C01669=1036.424,311.659,378.524,171.703,43.759,158.444
C01670=1036.430,311.906,378.490,171.706,43.760,158.445
C01671=1036.438,312.154,378.457,171.711,43.762,158.446
C01672=1036.445,312.401,378.422,171.715,43.764,158.447
C01673=1036.452,312.649,378.388,171.720,43.765,158.447
C01674=1036.458,312.896,378.354,171.724,43.767,158.448
C01675=1036.465,313.144,378.320,171.729,43.768,158.449
C01676=1036.472,313.392,378.286,171.733,43.770,158.449
C01677=1036.479,313.639,378.251,171.738,43.771,158.450
C01678=1036.486,313.887,378.217,171.741,43.773,158.451
C01679=1036.492,314.134,378.183,171.746,43.775,158.452
C01680=1036.499,314.382,378.149,171.750,43.777,158.452
C01681=1036.506,314.629,378.115,171.755,43.778,158.453
C01682=1036.513,314.877,378.080,171.760,43.779,158.454
C01683=1036.520,315.124,378.046,171.764,43.781,158.455
C01684=1036.527,315.371,378.012,171.769,43.783,158.455
C01685=1036.534,315.619,377.977,171.773,43.785,158.456
C01686=1036.541,315.867,377.943,171.778,43.786,158.457
C01687=1036.548,316.114,377.908,171.782,43.788,158.458
C01688=1036.555,316.362,377.875,171.787,43.789,158.458
C01689=1036.561,316.609,377.840,171.791,43.791,158.459
C01690=1036.568,316.856,377.806,171.796,43.793,158.460
C01691=1036.576,317.103,377.771,171.800,43.795,158.461
C01692=1036.582,317.351,377.737,171.804,43.796,158.462
C01693=1036.590,317.598,377.702,171.809,43.798,158.462
C01694=1036.596,317.846,377.668,171.813,43.800,158.463
C01695=1036.604,318.093,377.633,171.818,43.802,158.464
C01696=1036.610,318.341,377.599,171.823,43.803,158.465
C01697=1036.618,318.589,377.565,171.827,43.805,158.466
C01698=1036.624,318.836,377.530,171.832,43.806,158.466
C01699=1036.632,319.084,377.495,171.836,43.808,158.467
C01700=1036.639,319.332,377.461,171.841,43.810,158.468
C01701=1036.646,319.579,377.426,171.846,43.811,158.469
C01702=1036.657,319.953,377.374,171.852,43.814,158.470
C01703=1036.668,320.328,377.321,171.860,43.817,158.471
C01704=1036.679,320.702,377.269,171.866,43.820,158.472
C01705=1036.690,321.076,377.217,171.874,43.822,158.473
C01706=1036.697,321.323,377.182,171.878,43.824,158.474
C01707=1036.704,321.571,377.148,171.883,43.826,158.475
C01708=1036.711,321.818,377.113,171.888,43.827,158.476
C01709=1036.718,322.065,377.078,171.893,43.829,158.477
C01710=1036.725,322.313,377.043,171.897,43.831,158.477
C01711=1036.733,322.561,377.009,171.902,43.832,158.478
C01712=1036.739,322.808,376.974,171.907,43.834,158.479
C01713=1036.747,323.056,376.939,171.911,43.836,158.480
C01714=1036.754,323.303,376.904,171.916,43.838,158.481
C01715=1036.762,323.551,376.869,171.921,43.840,158.482
C01716=1036.769,323.798,376.834,171.926,43.841,158.482
C01717=1036.776,324.045,376.800,171.930,43.843,158.483
C01718=1036.783,324.292,376.764,171.935,43.845,158.484
C01719=1036.791,324.540,376.729,171.940,43.847,158.485
C01720=1036.798,324.788,376.694,171.944,43.849,158.486
C01721=1036.805,325.035,376.660,171.949,43.850,158.486
C01722=1036.813,325.283,376.624,171.954,43.852,158.487
C01723=1036.820,325.530,376.590,171.959,43.854,158.488
C01724=1036.827,325.777,376.555,171.964,43.856,158.489
C01725=1036.835,326.025,376.520,171.968,43.858,158.490
C01726=1036.842,326.272,376.485,171.973,43.859,158.491
C01727=1036.849,326.520,376.449,171.978,43.861,158.491
C01728=1036.857,326.767,376.415,171.983,43.863,158.492
C01729=1036.863,327.015,376.379,171.987,43.865,158.493
C01730=1036.872,327.262,376.344,171.992,43.867,158.494
C01731=1036.878,327.510,376.309,171.997,43.869,158.495
C01732=1036.886,327.758,376.274,172.002,43.871,158.496
C01733=1036.893,328.004,376.239,172.007,43.872,158.497
C01734=1036.901,328.251,376.204,172.012,43.875,158.497
C01735=1036.908,328.499,376.169,172.016,43.876,158.498
C01736=1036.915,328.747,376.133,172.021,43.879,158.499
C01737=1036.923,328.994,376.097,172.026,43.880,158.500
C01738=1036.930,329.242,376.062,172.032,43.882,158.501
C01739=1036.937,329.488,376.026,172.037,43.884,158.502
C01740=1036.945,329.736,375.991,172.041,43.886,158.503
C01741=1036.952,329.983,375.955,172.046,43.889,158.504
C01742=1036.959,330.231,375.920,172.051,43.890,158.505
C01743=1036.966,330.478,375.884,172.056,43.893,158.505
C01744=1036.974,330.726,375.849,172.061,43.894,158.506
C01745=1036.981,330.972,375.813,172.066,43.896,158.507
C01746=1036.988,331.221,375.777,172.070,43.899,158.508
C01747=1036.995,331.467,375.741,172.075,43.900,158.509
C01748=1037.002,331.715,375.706,172.081,43.903,158.510
C01749=1037.010,331.962,375.670,172.086,43.905,158.511
C01750=1037.017,332.210,375.634,172.091,43.907,158.512
C01751=1037.024,332.457,375.599,172.096,43.909,158.513
C01752=1037.032,332.704,375.562,172.101,43.911,158.514
C01753=1037.039,332.951,375.527,172.105,43.913,158.515
C01754=1037.046,333.199,375.491,172.110,43.915,158.515
C01755=1037.054,333.447,375.455,172.116,43.917,158.516
C01756=1037.061,333.693,375.419,172.121,43.919,158.517
C01757=1037.068,333.941,375.384,172.126,43.922,158.518
C01758=1037.079,334.311,375.330,172.134,43.925,158.520
C01759=1037.091,334.681,375.276,172.141,43.928,158.521
C01760=1037.102,335.050,375.223,172.149,43.931,158.522
C01761=1037.112,335.419,375.169,172.156,43.935,158.524
C01762=1037.120,335.667,375.132,172.161,43.937,158.525
C01763=1037.127,335.913,375.097,172.167,43.939,158.526
C01764=1037.134,336.161,375.060,172.172,43.941,158.527
C01765=1037.142,336.409,375.024,172.177,43.943,158.528
C01766=1037.149,336.655,374.988,172.182,43.946,158.529
C01767=1037.156,336.903,374.951,172.187,43.948,158.530
C01768=1037.163,337.151,374.915,172.193,43.950,158.531
C01769=1037.171,337.397,374.878,172.198,43.952,158.532
C01770=1037.178,337.644,374.842,172.203,43.954,158.533
C01771=1037.186,337.892,374.806,172.208,43.957,158.534
C01772=1037.194,338.139,374.769,172.213,43.959,158.535
C01773=1037.201,338.387,374.733,172.219,43.961,158.536
C01774=1037.208,338.634,374.697,172.224,43.963,158.537
C01775=1037.215,338.881,374.661,172.229,43.965,158.538
C01776=1037.223,339.128,374.624,172.235,43.968,158.539
C01777=1037.230,339.376,374.587,172.240,43.971,158.540
C01778=1037.238,339.623,374.551,172.245,43.973,158.541
C01779=1037.245,339.870,374.515,172.250,43.975,158.542
C01780=1037.253,340.117,374.478,172.255,43.977,158.543
C01781=1037.260,340.364,374.441,172.261,43.980,158.544
C01782=1037.268,340.612,374.405,172.266,43.982,158.545
C01783=1037.276,340.859,374.368,172.271,43.984,158.546
C01784=1037.283,341.106,374.332,172.277,43.987,158.547
C01785=1037.291,341.353,374.294,172.282,43.989,158.548
C01786=1037.298,341.600,374.258,172.287,43.991,158.549
C01787=1037.305,341.847,374.221,172.292,43.994,158.550
C01788=1037.313,342.095,374.184,172.298,43.996,158.551
C01789=1037.320,342.342,374.147,172.303,43.999,158.552
C01790=1037.327,342.589,374.111,172.309,44.001,158.553
C01791=1037.335,342.836,374.073,172.315,44.003,158.554
C01792=1037.342,343.084,374.037,172.320,44.006,158.555
C01793=1037.350,343.331,373.999,172.325,44.008,158.556
C01794=1037.358,343.578,373.963,172.331,44.011,158.557
C01795=1037.365,343.825,373.926,172.336,44.013,158.558
C01796=1037.372,344.072,373.889,172.341,44.016,158.559
C01797=1037.380,344.319,373.851,172.347,44.018,158.561
C01798=1037.388,344.566,373.814,172.352,44.021,158.561
C01799=1037.395,344.814,373.778,172.357,44.023,158.563
C01800=1037.403,345.061,373.741,172.364,44.026,158.564
C01801=1037.410,345.308,373.703,172.369,44.028,158.565
C01802=1037.418,345.555,373.666,172.375,44.031,158.566
C01803=1037.425,345.802,373.629,172.380,44.033,158.567
C01804=1037.433,346.049,373.592,172.385,44.036,158.568
C01805=1037.440,346.296,373.555,172.391,44.039,158.569
C01806=1037.447,346.544,373.517,172.396,44.041,158.570
C01807=1037.455,346.790,373.480,172.402,44.043,158.571
C01808=1037.463,347.038,373.443,172.408,44.046,158.573
C01809=1037.470,347.284,373.406,172.413,44.049,158.574
C01810=1037.478,347.531,373.368,172.419,44.051,158.575
C01811=1037.486,347.779,373.331,172.424,44.054,158.576
C01812=1037.494,348.026,373.294,172.431,44.057,158.577
C01813=1037.501,348.273,373.256,172.436,44.059,158.578
C01814=1037.513,348.639,373.200,172.444,44.063,158.580
C01815=1037.524,349.005,373.145,172.452,44.067,158.581
C01816=1037.535,349.371,373.089,172.461,44.071,158.583
C01817=1037.546,349.738,373.034,172.470,44.075,158.585
